LIN {X 0,Y 409.998,Z 362.021,A -85,B 0,C 180,E1 -10362.384,E2 -10362.384} C_VEL
LIN {X 0,Y 409.907,Z 362.961,A -85,B 0,C 180,E1 -10363.887,E2 -10363.887} C_VEL
LIN {X 0,Y 409.94,Z 362.921,A -85,B 0,C 180,E1 -10364.9,E2 -10364.9} C_VEL
LIN {X 0,Y 410.047,Z 362.009,A -85,B 0,C 180,E1 -10366.309,E2 -10366.309} C_VEL
LIN {X 0,Y 410.116,Z 361.339,A -85,B 0,C 180,E1 -10366.936,E2 -10366.936} C_VEL
LIN {X 0,Y 410.312,Z 358.576,A -85,B 0,C 180,E1 -10368.473,E2 -10368.473} C_VEL
LIN {X 0,Y 410.578,Z 355.393,A -85,B 0,C 180,E1 -10369.711,E2 -10369.711} C_VEL
LIN {X 0,Y 410.758,Z 352.823,A -85,B 0,C 180,E1 -10370.532,E2 -10370.532} C_VEL
LIN {X 0,Y 411.107,Z 347.629,A -85,B 0,C 180,E1 -10371.826,E2 -10371.826} C_VEL
LIN {X 0,Y 411.62,Z 341.02,A -85,B 0,C 180,E1 -10373.121,E2 -10373.121} C_VEL
LIN {X 0,Y 412.051,Z 334.444,A -85,B 0,C 180,E1 -10374.162,E2 -10374.162} C_VEL
LIN {X 0,Y 412.673,Z 326.386,A -85,B 0,C 180,E1 -10375.197,E2 -10375.197} C_VEL
LIN {X 0,Y 413.3,Z 315.956,A -85,B 0,C 180,E1 -10376.238,E2 -10376.238} C_VEL
LIN {X 0,Y 413.735,Z 307.563,A -85,B 0,C 180,E1 -10376.888,E2 -10376.888} C_VEL
LIN {X 0,Y 413.706,Z 301.383,A -85,B 0,C 180,E1 -10377.3,E2 -10377.3} C_VEL
LIN {X 0,Y 411.503,Z 290.548,A -85,B 0,C 180,E1 -10377.925,E2 -10377.925} C_VEL
LIN {X 0,Y 410.193,Z 285.02,A -85,B 0,C 180,E1 -10378.2,E2 -10378.2} C_VEL
LIN {X 0,Y 410.313,Z 281.535,A -85,B 0,C 180,E1 -10381.088,E2 -10381.088} C_VEL
LIN {X 0,Y 410.369,Z 277.277,A -85,B 0,C 180,E1 -10384.714,E2 -10384.714} C_VEL
LIN {X 0,Y 410.554,Z 273.44,A -85,B 0,C 180,E1 -10388.057,E2 -10388.057} C_VEL
LIN {X 0,Y 410.699,Z 269.952,A -85,B 0,C 180,E1 -10391.158,E2 -10391.158} C_VEL
LIN {X 0,Y 410.819,Z 266.266,A -85,B 0,C 180,E1 -10394.537,E2 -10394.537} C_VEL
LIN {X 0,Y 411.08,Z 266.09,A -85,B 0,C 180,E1 -10397.317,E2 -10397.317} C_VEL
LIN {X 0,Y 411.211,Z 266.076,A -85,B 0,C 180,E1 -10400.778,E2 -10400.778} C_VEL
LIN {X 0,Y 411.18,Z 266.082,A -85,B 0,C 180,E1 -10404.473,E2 -10404.473} C_VEL
LIN {X 0,Y 411.188,Z 266.079,A -85,B 0,C 180,E1 -10406.874,E2 -10406.874} C_VEL
LIN {X 0,Y 411.214,Z 266.077,A -85,B 0,C 180,E1 -10410.645,E2 -10410.645} C_VEL
LIN {X 0,Y 411.219,Z 266.075,A -85,B 0,C 180,E1 -10413.62,E2 -10413.62} C_VEL
LIN {X 0,Y 411.179,Z 266.08,A -85,B 0,C 180,E1 -10416.853,E2 -10416.853} C_VEL
LIN {X 0,Y 411.199,Z 266.078,A -85,B 0,C 180,E1 -10420.052,E2 -10420.052} C_VEL
LIN {X 0,Y 411.247,Z 266.07,A -85,B 0,C 180,E1 -10423.133,E2 -10423.133} C_VEL
LIN {X 0,Y 411.299,Z 266.064,A -85,B 0,C 180,E1 -10426.893,E2 -10426.893} C_VEL
LIN {X 0,Y 411.295,Z 266.063,A -85,B 0,C 180,E1 -10430.163,E2 -10430.163} C_VEL
LIN {X 0,Y 411.41,Z 266.047,A -85,B 0,C 180,E1 -10433.134,E2 -10433.134} C_VEL
LIN {X 0,Y 411.457,Z 266.044,A -85,B 0,C 180,E1 -10437.065,E2 -10437.065} C_VEL
LIN {X 0,Y 411.629,Z 266.022,A -85,B 0,C 180,E1 -10440.002,E2 -10440.002} C_VEL
LIN {X 0,Y 411.447,Z 266.044,A -85,B 0,C 180,E1 -10442.939,E2 -10442.939} C_VEL
LIN {X 0,Y 411.451,Z 266.044,A -85,B 0,C 180,E1 -10446.869,E2 -10446.869} C_VEL
LIN {X 0,Y 411.285,Z 266.066,A -85,B 0,C 180,E1 -10449.841,E2 -10449.841} C_VEL
LIN {X 0,Y 411.304,Z 266.065,A -85,B 0,C 180,E1 -10453.111,E2 -10453.111} C_VEL
LIN {X 0,Y 411.249,Z 266.071,A -85,B 0,C 180,E1 -10456.891,E2 -10456.891} C_VEL
LIN {X 0,Y 411.223,Z 266.075,A -85,B 0,C 180,E1 -10459.989,E2 -10459.989} C_VEL
LIN {X 0,Y 411.189,Z 266.08,A -85,B 0,C 180,E1 -10463.15,E2 -10463.15} C_VEL
LIN {X 0,Y 411.189,Z 266.081,A -85,B 0,C 180,E1 -10466.386,E2 -10466.386} C_VEL
LIN {X 0,Y 411.192,Z 266.081,A -85,B 0,C 180,E1 -10469.715,E2 -10469.715} C_VEL
LIN {X 0,Y 411.201,Z 266.08,A -85,B 0,C 180,E1 -10473.158,E2 -10473.158} C_VEL
LIN {X 0,Y 411.187,Z 266.081,A -85,B 0,C 180,E1 -10476.554,E2 -10476.554} C_VEL
LIN {X 0,Y 411.222,Z 266.075,A -85,B 0,C 180,E1 -10479.732,E2 -10479.732} C_VEL
LIN {X 0,Y 411.173,Z 266.083,A -85,B 0,C 180,E1 -10483.135,E2 -10483.135} C_VEL
LIN {X 0,Y 411.164,Z 266.082,A -85,B 0,C 180,E1 -10485.883,E2 -10485.883} C_VEL
LIN {X 0,Y 411.16,Z 266.085,A -85,B 0,C 180,E1 -10488.774,E2 -10488.774} C_VEL
LIN {X 0,Y 411.218,Z 266.113,A -85,B 0,C 180,E1 -10490.778,E2 -10490.778} C_VEL
LIN {X 0,Y 412.203,Z 271.693,A -85,B 0,C 180,E1 -10493.971,E2 -10493.971} C_VEL
LIN {X 0,Y 412.916,Z 276.371,A -85,B 0,C 180,E1 -10496.513,E2 -10496.513} C_VEL
LIN {X 0,Y 412.699,Z 280.103,A -85,B 0,C 180,E1 -10498.373,E2 -10498.373} C_VEL
LIN {X 0,Y 412.092,Z 286.591,A -85,B 0,C 180,E1 -10501.478,E2 -10501.478} C_VEL
LIN {X 0,Y 411.4,Z 294.979,A -85,B 0,C 180,E1 -10505.329,E2 -10505.329} C_VEL
LIN {X 0,Y 410.851,Z 303.168,A -85,B 0,C 180,E1 -10508.949,E2 -10508.949} C_VEL
LIN {X 0,Y 410.524,Z 311.551,A -85,B 0,C 180,E1 -10512.568,E2 -10512.568} C_VEL
LIN {X 0,Y 410.219,Z 319.243,A -85,B 0,C 180,E1 -10515.807,E2 -10515.807} C_VEL
LIN {X 0,Y 411.907,Z 330.548,A -85,B 0,C 180,E1 -10516.284,E2 -10516.284} C_VEL
LIN {X 0,Y 412.841,Z 341.087,A -85,B 0,C 180,E1 -10516.9,E2 -10516.9} C_VEL
LIN {X 0,Y 412.852,Z 349.045,A -85,B 0,C 180,E1 -10517.466,E2 -10517.466} C_VEL
LIN {X 0,Y 412.264,Z 357.493,A -85,B 0,C 180,E1 -10518.197,E2 -10518.197} C_VEL
LIN {X 0,Y 411.762,Z 365.475,A -85,B 0,C 180,E1 -10519.055,E2 -10519.055} C_VEL
LIN {X 0,Y 411.295,Z 372.086,A -85,B 0,C 180,E1 -10519.914,E2 -10519.914} C_VEL
LIN {X 0,Y 410.86,Z 378.38,A -85,B 0,C 180,E1 -10520.897,E2 -10520.897} C_VEL
LIN {X 0,Y 410.538,Z 383.622,A -85,B 0,C 180,E1 -10521.882,E2 -10521.882} C_VEL
LIN {X 0,Y 410.251,Z 388.968,A -85,B 0,C 180,E1 -10523.114,E2 -10523.114} C_VEL
LIN {X 0,Y 410.082,Z 392.428,A -85,B 0,C 180,E1 -10524.099,E2 -10524.099} C_VEL
LIN {X 0,Y 410.021,Z 396.434,A -85,B 0,C 180,E1 -10525.578,E2 -10525.578} C_VEL
LIN {X 0,Y 409.985,Z 399.189,A -85,B 0,C 180,E1 -10527.054,E2 -10527.054} C_VEL
LIN {X 0,Y 410.021,Z 400.293,A -85,B 0,C 180,E1 -10528.037,E2 -10528.037} C_VEL
LIN {X 0,Y 409.979,Z 400.923,A -85,B 0,C 180,E1 -10529.019,E2 -10529.019} C_VEL
LIN {X 0,Y 409.974,Z 401.092,A -85,B 0,C 180,E1 -10530.001,E2 -10530.001} C_VEL
LIN {X 0,Y 409.979,Z 400.763,A -85,B 0,C 180,E1 -10530.984,E2 -10530.984} C_VEL
LIN {X 0,Y 410.025,Z 399.839,A -85,B 0,C 180,E1 -10531.966,E2 -10531.966} C_VEL
LIN {X 0,Y 410.021,Z 398.414,A -85,B 0,C 180,E1 -10532.949,E2 -10532.949} C_VEL
LIN {X 0,Y 410.022,Z 395.317,A -85,B 0,C 180,E1 -10534.425,E2 -10534.425} C_VEL
LIN {X 0,Y 410.068,Z 390.877,A -85,B 0,C 180,E1 -10535.903,E2 -10535.903} C_VEL
LIN {X 0,Y 410.334,Z 385.927,A -85,B 0,C 180,E1 -10537.134,E2 -10537.134} C_VEL
LIN {X 0,Y 410.538,Z 379.661,A -85,B 0,C 180,E1 -10538.368,E2 -10538.368} C_VEL
LIN {X 0,Y 410.816,Z 373.538,A -85,B 0,C 180,E1 -10539.354,E2 -10539.354} C_VEL
LIN {X 0,Y 411.261,Z 366.093,A -85,B 0,C 180,E1 -10540.338,E2 -10540.338} C_VEL
LIN {X 0,Y 411.655,Z 358.104,A -85,B 0,C 180,E1 -10541.199,E2 -10541.199} C_VEL
LIN {X 0,Y 412.187,Z 348.138,A -85,B 0,C 180,E1 -10542.057,E2 -10542.057} C_VEL
LIN {X 0,Y 411.964,Z 338.649,A -85,B 0,C 180,E1 -10542.689,E2 -10542.689} C_VEL
LIN {X 0,Y 411.03,Z 328.221,A -85,B 0,C 180,E1 -10543.212,E2 -10543.212} C_VEL
LIN {X 0,Y 410.158,Z 319.531,A -85,B 0,C 180,E1 -10543.534,E2 -10543.534} C_VEL
LIN {X 0,Y 410.403,Z 311.332,A -85,B 0,C 180,E1 -10546.926,E2 -10546.926} C_VEL
LIN {X 0,Y 410.692,Z 302.714,A -85,B 0,C 180,E1 -10550.538,E2 -10550.538} C_VEL
LIN {X 0,Y 411.06,Z 295.284,A -85,B 0,C 180,E1 -10553.691,E2 -10553.691} C_VEL
LIN {X 0,Y 411.607,Z 286.782,A -85,B 0,C 180,E1 -10557.391,E2 -10557.391} C_VEL
LIN {X 0,Y 412.159,Z 279.227,A -85,B 0,C 180,E1 -10560.768,E2 -10560.768} C_VEL
LIN {X 0,Y 412.454,Z 273.561,A -85,B 0,C 180,E1 -10563.39,E2 -10563.39} C_VEL
LIN {X 0,Y 411.599,Z 268.219,A -85,B 0,C 180,E1 -10566.027,E2 -10566.027} C_VEL
LIN {X 0,Y 411.234,Z 266.075,A -85,B 0,C 180,E1 -10567.198,E2 -10567.198} C_VEL
LIN {X 0,Y 411.188,Z 266.079,A -85,B 0,C 180,E1 -10570.505,E2 -10570.505} C_VEL
LIN {X 0,Y 411.182,Z 266.078,A -85,B 0,C 180,E1 -10573.134,E2 -10573.134} C_VEL
LIN {X 0,Y 411.177,Z 266.082,A -85,B 0,C 180,E1 -10575.881,E2 -10575.881} C_VEL
LIN {X 0,Y 411.172,Z 266.079,A -85,B 0,C 180,E1 -10578.772,E2 -10578.772} C_VEL
LIN {X 0,Y 411.198,Z 266.079,A -85,B 0,C 180,E1 -10582.025,E2 -10582.025} C_VEL
LIN {X 0,Y 411.215,Z 266.078,A -85,B 0,C 180,E1 -10585.666,E2 -10585.666} C_VEL
LIN {X 0,Y 411.199,Z 266.078,A -85,B 0,C 180,E1 -10589.152,E2 -10589.152} C_VEL
LIN {X 0,Y 411.268,Z 266.067,A -85,B 0,C 180,E1 -10592.522,E2 -10592.522} C_VEL
LIN {X 0,Y 411.229,Z 266.074,A -85,B 0,C 180,E1 -10595.783,E2 -10595.783} C_VEL
LIN {X 0,Y 411.205,Z 266.079,A -85,B 0,C 180,E1 -10598.965,E2 -10598.965} C_VEL
LIN {X 0,Y 411.254,Z 266.069,A -85,B 0,C 180,E1 -10602.084,E2 -10602.084} C_VEL
LIN {X 0,Y 411.268,Z 266.071,A -85,B 0,C 180,E1 -10605.146,E2 -10605.146} C_VEL
LIN {X 0,Y 411.291,Z 266.065,A -85,B 0,C 180,E1 -10608.166,E2 -10608.166} C_VEL
LIN {X 0,Y 411.446,Z 266.046,A -85,B 0,C 180,E1 -10612.19,E2 -10612.19} C_VEL
LIN {X 0,Y 411.473,Z 266.043,A -85,B 0,C 180,E1 -10614.116,E2 -10614.116} C_VEL
LIN {X 0,Y 411.517,Z 266.037,A -85,B 0,C 180,E1 -10618.041,E2 -10618.041} C_VEL
LIN {X 0,Y 411.646,Z 266.021,A -85,B 0,C 180,E1 -10619.998,E2 -10619.998} C_VEL
LIN {X 0,Y 411.47,Z 266.044,A -85,B 0,C 180,E1 -10622.935,E2 -10622.935} C_VEL
LIN {X 0,Y 411.465,Z 266.045,A -85,B 0,C 180,E1 -10626.865,E2 -10626.865} C_VEL
LIN {X 0,Y 411.358,Z 266.058,A -85,B 0,C 180,E1 -10628.843,E2 -10628.843} C_VEL
LIN {X 0,Y 411.287,Z 266.067,A -85,B 0,C 180,E1 -10631.831,E2 -10631.831} C_VEL
LIN {X 0,Y 411.262,Z 266.069,A -85,B 0,C 180,E1 -10634.85,E2 -10634.85} C_VEL
LIN {X 0,Y 411.254,Z 266.072,A -85,B 0,C 180,E1 -10637.913,E2 -10637.913} C_VEL
LIN {X 0,Y 411.197,Z 266.076,A -85,B 0,C 180,E1 -10641.032,E2 -10641.032} C_VEL
LIN {X 0,Y 411.226,Z 266.075,A -85,B 0,C 180,E1 -10644.213,E2 -10644.213} C_VEL
LIN {X 0,Y 411.257,Z 266.072,A -85,B 0,C 180,E1 -10647.475,E2 -10647.475} C_VEL
LIN {X 0,Y 411.186,Z 266.077,A -85,B 0,C 180,E1 -10650.845,E2 -10650.845} C_VEL
LIN {X 0,Y 411.202,Z 266.076,A -85,B 0,C 180,E1 -10654.331,E2 -10654.331} C_VEL
LIN {X 0,Y 411.199,Z 266.078,A -85,B 0,C 180,E1 -10657.97,E2 -10657.97} C_VEL
LIN {X 0,Y 411.203,Z 266.079,A -85,B 0,C 180,E1 -10661.233,E2 -10661.233} C_VEL
LIN {X 0,Y 411.229,Z 266.073,A -85,B 0,C 180,E1 -10664.48,E2 -10664.48} C_VEL
LIN {X 0,Y 411.22,Z 266.077,A -85,B 0,C 180,E1 -10667.295,E2 -10667.295} C_VEL
LIN {X 0,Y 411.222,Z 266.076,A -85,B 0,C 180,E1 -10670.775,E2 -10670.775} C_VEL
LIN {X 0,Y 411.188,Z 266.078,A -85,B 0,C 180,E1 -10674.469,E2 -10674.469} C_VEL
LIN {X 0,Y 411.195,Z 266.08,A -85,B 0,C 180,E1 -10676.871,E2 -10676.871} C_VEL
LIN {X 0,Y 411.228,Z 266.076,A -85,B 0,C 180,E1 -10680.64,E2 -10680.64} C_VEL
LIN {X 0,Y 411.224,Z 266.073,A -85,B 0,C 180,E1 -10683.617,E2 -10683.617} C_VEL
LIN {X 0,Y 411.194,Z 266.079,A -85,B 0,C 180,E1 -10686.851,E2 -10686.851} C_VEL
LIN {X 0,Y 411.199,Z 266.078,A -85,B 0,C 180,E1 -10690.048,E2 -10690.048} C_VEL
LIN {X 0,Y 410.957,Z 266.107,A -85,B 0,C 180,E1 -10693.263,E2 -10693.263} C_VEL
LIN {X 0,Y 410.693,Z 266.143,A -85,B 0,C 180,E1 -10695.125,E2 -10695.125} C_VEL
LIN {X 0,Y 410.71,Z 268.309,A -85,B 0,C 180,E1 -10697.245,E2 -10697.245} C_VEL
LIN {X 0,Y 410.537,Z 272.981,A -85,B 0,C 180,E1 -10701.136,E2 -10701.136} C_VEL
LIN {X 0,Y 410.601,Z 275.356,A -85,B 0,C 180,E1 -10703.117,E2 -10703.117} C_VEL
LIN {X 0,Y 410.49,Z 278.995,A -85,B 0,C 180,E1 -10706.072,E2 -10706.072} C_VEL
LIN {X 0,Y 410.232,Z 282.687,A -85,B 0,C 180,E1 -10709.017,E2 -10709.017} C_VEL
LIN {X 0,Y 410.145,Z 284.671,A -85,B 0,C 180,E1 -10710.582,E2 -10710.582} C_VEL
LIN {X 0,Y 412.205,Z 296.714,A -85,B 0,C 180,E1 -10711.159,E2 -10711.159} C_VEL
LIN {X 0,Y 412.893,Z 302.077,A -85,B 0,C 180,E1 -10711.462,E2 -10711.462} C_VEL
LIN {X 0,Y 412.472,Z 312.617,A -85,B 0,C 180,E1 -10712.196,E2 -10712.196} C_VEL
LIN {X 0,Y 412.107,Z 320.89,A -85,B 0,C 180,E1 -10712.931,E2 -10712.931} C_VEL
LIN {X 0,Y 411.672,Z 328.745,A -85,B 0,C 180,E1 -10713.792,E2 -10713.792} C_VEL
LIN {X 0,Y 411.389,Z 335.207,A -85,B 0,C 180,E1 -10714.653,E2 -10714.653} C_VEL
LIN {X 0,Y 410.976,Z 341.39,A -85,B 0,C 180,E1 -10715.642,E2 -10715.642} C_VEL
LIN {X 0,Y 410.771,Z 347.667,A -85,B 0,C 180,E1 -10716.877,E2 -10716.877} C_VEL
LIN {X 0,Y 410.391,Z 353.532,A -85,B 0,C 180,E1 -10718.369,E2 -10718.369} C_VEL
LIN {X 0,Y 410.237,Z 356.577,A -85,B 0,C 180,E1 -10719.365,E2 -10719.365} C_VEL
LIN {X 0,Y 410.083,Z 359.907,A -85,B 0,C 180,E1 -10720.865,E2 -10720.865} C_VEL
LIN {X 0,Y 410.006,Z 361.951,A -85,B 0,C 180,E1 -10722.313,E2 -10722.313} C_VEL
LIN {X 0,Y 409.998,Z 362.021,A -85,B 0,C 180,E1 -10722.384,E2 -10722.384} C_VEL
LIN {X 0,Y 409.271,Z 362.759,A -85,B 0,C 180,E1 -10723.2,E2 -10723.2} C_VEL
LIN {X 0,Y 406.381,Z 363.211,A -85,B 0,C 180,E1 -10724.532,E2 -10724.532} C_VEL
LIN {X 0,Y 403.577,Z 362.803,A -85,B 0,C 180,E1 -10725.882,E2 -10725.882} C_VEL
LIN {X 0,Y 402.999,Z 361.972,A -85,B 0,C 180,E1 -10726.713,E2 -10726.713} C_VEL
LIN {X 0,Y 403.203,Z 359.617,A -85,B 0,C 180,E1 -10728.284,E2 -10728.284} C_VEL
LIN {X 0,Y 403.416,Z 357.245,A -85,B 0,C 180,E1 -10729.328,E2 -10729.328} C_VEL
LIN {X 0,Y 403.766,Z 352.366,A -85,B 0,C 180,E1 -10730.904,E2 -10730.904} C_VEL
LIN {X 0,Y 404.11,Z 348.209,A -85,B 0,C 180,E1 -10731.956,E2 -10731.956} C_VEL
LIN {X 0,Y 404.606,Z 342.156,A -85,B 0,C 180,E1 -10733.183,E2 -10733.183} C_VEL
LIN {X 0,Y 405.012,Z 336.926,A -85,B 0,C 180,E1 -10734.064,E2 -10734.064} C_VEL
LIN {X 0,Y 405.465,Z 330.348,A -85,B 0,C 180,E1 -10734.991,E2 -10734.991} C_VEL
LIN {X 0,Y 405.972,Z 323.212,A -85,B 0,C 180,E1 -10735.822,E2 -10735.822} C_VEL
LIN {X 0,Y 406.504,Z 315.296,A -85,B 0,C 180,E1 -10736.577,E2 -10736.577} C_VEL
LIN {X 0,Y 406.915,Z 307.924,A -85,B 0,C 180,E1 -10737.152,E2 -10737.152} C_VEL
LIN {X 0,Y 406.94,Z 302.908,A -85,B 0,C 180,E1 -10737.498,E2 -10737.498} C_VEL
LIN {X 0,Y 404.603,Z 291.351,A -85,B 0,C 180,E1 -10738.2,E2 -10738.2} C_VEL
LIN {X 0,Y 403.15,Z 285.374,A -85,B 0,C 180,E1 -10738.504,E2 -10738.504} C_VEL
LIN {X 0,Y 403.26,Z 281.77,A -85,B 0,C 180,E1 -10741.521,E2 -10741.521} C_VEL
LIN {X 0,Y 403.314,Z 277.633,A -85,B 0,C 180,E1 -10745.101,E2 -10745.101} C_VEL
LIN {X 0,Y 403.506,Z 273.912,A -85,B 0,C 180,E1 -10748.397,E2 -10748.397} C_VEL
LIN {X 0,Y 403.662,Z 270.44,A -85,B 0,C 180,E1 -10751.53,E2 -10751.53} C_VEL
LIN {X 0,Y 403.79,Z 267.269,A -85,B 0,C 180,E1 -10754.474,E2 -10754.474} C_VEL
LIN {X 0,Y 404.016,Z 266.97,A -85,B 0,C 180,E1 -10756.935,E2 -10756.935} C_VEL
LIN {X 0,Y 404.148,Z 266.956,A -85,B 0,C 180,E1 -10759.956,E2 -10759.956} C_VEL
LIN {X 0,Y 404.121,Z 266.961,A -85,B 0,C 180,E1 -10763.125,E2 -10763.125} C_VEL
LIN {X 0,Y 404.126,Z 266.96,A -85,B 0,C 180,E1 -10766.189,E2 -10766.189} C_VEL
LIN {X 0,Y 404.127,Z 266.957,A -85,B 0,C 180,E1 -10769.716,E2 -10769.716} C_VEL
LIN {X 0,Y 404.177,Z 266.951,A -85,B 0,C 180,E1 -10773.124,E2 -10773.124} C_VEL
LIN {X 0,Y 404.157,Z 266.956,A -85,B 0,C 180,E1 -10775.336,E2 -10775.336} C_VEL
LIN {X 0,Y 404.122,Z 266.958,A -85,B 0,C 180,E1 -10778.582,E2 -10778.582} C_VEL
LIN {X 0,Y 404.194,Z 266.949,A -85,B 0,C 180,E1 -10781.763,E2 -10781.763} C_VEL
LIN {X 0,Y 404.192,Z 266.95,A -85,B 0,C 180,E1 -10784.884,E2 -10784.884} C_VEL
LIN {X 0,Y 404.256,Z 266.945,A -85,B 0,C 180,E1 -10787.961,E2 -10787.961} C_VEL
LIN {X 0,Y 404.281,Z 266.939,A -85,B 0,C 180,E1 -10791.001,E2 -10791.001} C_VEL
LIN {X 0,Y 404.379,Z 266.923,A -85,B 0,C 180,E1 -10794.016,E2 -10794.016} C_VEL
LIN {X 0,Y 404.472,Z 266.912,A -85,B 0,C 180,E1 -10798.01,E2 -10798.01} C_VEL
LIN {X 0,Y 404.599,Z 266.898,A -85,B 0,C 180,E1 -10800.002,E2 -10800.002} C_VEL
LIN {X 0,Y 404.405,Z 266.921,A -85,B 0,C 180,E1 -10802.99,E2 -10802.99} C_VEL
LIN {X 0,Y 404.402,Z 266.923,A -85,B 0,C 180,E1 -10806.989,E2 -10806.989} C_VEL
LIN {X 0,Y 404.251,Z 266.944,A -85,B 0,C 180,E1 -10810.013,E2 -10810.013} C_VEL
LIN {X 0,Y 404.257,Z 266.943,A -85,B 0,C 180,E1 -10813.213,E2 -10813.213} C_VEL
LIN {X 0,Y 404.207,Z 266.948,A -85,B 0,C 180,E1 -10817.009,E2 -10817.009} C_VEL
LIN {X 0,Y 404.156,Z 266.953,A -85,B 0,C 180,E1 -10820.353,E2 -10820.353} C_VEL
LIN {X 0,Y 404.153,Z 266.954,A -85,B 0,C 180,E1 -10823.577,E2 -10823.577} C_VEL
LIN {X 0,Y 404.128,Z 266.959,A -85,B 0,C 180,E1 -10826.883,E2 -10826.883} C_VEL
LIN {X 0,Y 404.138,Z 266.959,A -85,B 0,C 180,E1 -10830.287,E2 -10830.287} C_VEL
LIN {X 0,Y 404.139,Z 266.963,A -85,B 0,C 180,E1 -10833.814,E2 -10833.814} C_VEL
LIN {X 0,Y 404.132,Z 266.961,A -85,B 0,C 180,E1 -10836.877,E2 -10836.877} C_VEL
LIN {X 0,Y 404.161,Z 266.956,A -85,B 0,C 180,E1 -10840.085,E2 -10840.085} C_VEL
LIN {X 0,Y 404.154,Z 266.957,A -85,B 0,C 180,E1 -10843.086,E2 -10843.086} C_VEL
LIN {X 0,Y 404.144,Z 266.956,A -85,B 0,C 180,E1 -10845.928,E2 -10845.928} C_VEL
LIN {X 0,Y 404.115,Z 266.963,A -85,B 0,C 180,E1 -10848.637,E2 -10848.637} C_VEL
LIN {X 0,Y 404.185,Z 267.016,A -85,B 0,C 180,E1 -10850.446,E2 -10850.446} C_VEL
LIN {X 0,Y 405.207,Z 272.822,A -85,B 0,C 180,E1 -10853.866,E2 -10853.866} C_VEL
LIN {X 0,Y 405.893,Z 277.333,A -85,B 0,C 180,E1 -10856.355,E2 -10856.355} C_VEL
LIN {X 0,Y 405.601,Z 281.932,A -85,B 0,C 180,E1 -10858.682,E2 -10858.682} C_VEL
LIN {X 0,Y 405.067,Z 287.708,A -85,B 0,C 180,E1 -10861.504,E2 -10861.504} C_VEL
LIN {X 0,Y 404.342,Z 295.939,A -85,B 0,C 180,E1 -10865.347,E2 -10865.347} C_VEL
LIN {X 0,Y 403.781,Z 304.226,A -85,B 0,C 180,E1 -10869.097,E2 -10869.097} C_VEL
LIN {X 0,Y 403.427,Z 312.579,A -85,B 0,C 180,E1 -10872.775,E2 -10872.775} C_VEL
LIN {X 0,Y 403.19,Z 318.864,A -85,B 0,C 180,E1 -10875.49,E2 -10875.49} C_VEL
LIN {X 0,Y 405.072,Z 331.754,A -85,B 0,C 180,E1 -10876.079,E2 -10876.079} C_VEL
LIN {X 0,Y 405.926,Z 341.516,A -85,B 0,C 180,E1 -10876.677,E2 -10876.677} C_VEL
LIN {X 0,Y 405.937,Z 349.273,A -85,B 0,C 180,E1 -10877.249,E2 -10877.249} C_VEL
LIN {X 0,Y 405.333,Z 357.62,A -85,B 0,C 180,E1 -10877.992,E2 -10877.992} C_VEL
LIN {X 0,Y 404.803,Z 365.524,A -85,B 0,C 180,E1 -10878.865,E2 -10878.865} C_VEL
LIN {X 0,Y 404.312,Z 372.071,A -85,B 0,C 180,E1 -10879.738,E2 -10879.738} C_VEL
LIN {X 0,Y 403.849,Z 378.313,A -85,B 0,C 180,E1 -10880.738,E2 -10880.738} C_VEL
LIN {X 0,Y 403.48,Z 383.508,A -85,B 0,C 180,E1 -10881.739,E2 -10881.739} C_VEL
LIN {X 0,Y 403.19,Z 388.81,A -85,B 0,C 180,E1 -10882.993,E2 -10882.993} C_VEL
LIN {X 0,Y 402.981,Z 393.763,A -85,B 0,C 180,E1 -10884.497,E2 -10884.497} C_VEL
LIN {X 0,Y 402.893,Z 397.281,A -85,B 0,C 180,E1 -10886,E2 -10886} C_VEL
LIN {X 0,Y 402.884,Z 398.926,A -85,B 0,C 180,E1 -10887.002,E2 -10887.002} C_VEL
LIN {X 0,Y 402.95,Z 400.003,A -85,B 0,C 180,E1 -10888.002,E2 -10888.002} C_VEL
LIN {X 0,Y 402.904,Z 400.606,A -85,B 0,C 180,E1 -10889.002,E2 -10889.002} C_VEL
LIN {X 0,Y 402.896,Z 400.749,A -85,B 0,C 180,E1 -10890.001,E2 -10890.001} C_VEL
LIN {X 0,Y 402.904,Z 400.407,A -85,B 0,C 180,E1 -10891.001,E2 -10891.001} C_VEL
LIN {X 0,Y 402.954,Z 399.47,A -85,B 0,C 180,E1 -10892,E2 -10892} C_VEL
LIN {X 0,Y 402.92,Z 398.016,A -85,B 0,C 180,E1 -10893.001,E2 -10893.001} C_VEL
LIN {X 0,Y 402.952,Z 394.891,A -85,B 0,C 180,E1 -10894.503,E2 -10894.503} C_VEL
LIN {X 0,Y 402.991,Z 390.392,A -85,B 0,C 180,E1 -10896.008,E2 -10896.008} C_VEL
LIN {X 0,Y 403.281,Z 385.394,A -85,B 0,C 180,E1 -10897.26,E2 -10897.26} C_VEL
LIN {X 0,Y 403.497,Z 379.08,A -85,B 0,C 180,E1 -10898.515,E2 -10898.515} C_VEL
LIN {X 0,Y 403.782,Z 372.902,A -85,B 0,C 180,E1 -10899.519,E2 -10899.519} C_VEL
LIN {X 0,Y 404.192,Z 366.42,A -85,B 0,C 180,E1 -10900.394,E2 -10900.394} C_VEL
LIN {X 0,Y 404.495,Z 359.793,A -85,B 0,C 180,E1 -10901.146,E2 -10901.146} C_VEL
LIN {X 0,Y 404.986,Z 351.783,A -85,B 0,C 180,E1 -10901.894,E2 -10901.894} C_VEL
LIN {X 0,Y 405.217,Z 343.667,A -85,B 0,C 180,E1 -10902.509,E2 -10902.509} C_VEL
LIN {X 0,Y 404.553,Z 334.884,A -85,B 0,C 180,E1 -10903.053,E2 -10903.053} C_VEL
LIN {X 0,Y 403.724,Z 325.792,A -85,B 0,C 180,E1 -10903.484,E2 -10903.484} C_VEL
LIN {X 0,Y 403.086,Z 319.207,A -85,B 0,C 180,E1 -10903.74,E2 -10903.74} C_VEL
LIN {X 0,Y 403.323,Z 310.929,A -85,B 0,C 180,E1 -10907.232,E2 -10907.232} C_VEL
LIN {X 0,Y 403.65,Z 302.331,A -85,B 0,C 180,E1 -10910.913,E2 -10910.913} C_VEL
LIN {X 0,Y 403.983,Z 296.148,A -85,B 0,C 180,E1 -10913.587,E2 -10913.587} C_VEL
LIN {X 0,Y 404.45,Z 288.78,A -85,B 0,C 180,E1 -10916.86,E2 -10916.86} C_VEL
LIN {X 0,Y 405.032,Z 281.362,A -85,B 0,C 180,E1 -10920.213,E2 -10920.213} C_VEL
LIN {X 0,Y 405.448,Z 275.249,A -85,B 0,C 180,E1 -10923.081,E2 -10923.081} C_VEL
LIN {X 0,Y 404.836,Z 270.727,A -85,B 0,C 180,E1 -10925.32,E2 -10925.32} C_VEL
LIN {X 0,Y 404.171,Z 266.955,A -85,B 0,C 180,E1 -10927.323,E2 -10927.323} C_VEL
LIN {X 0,Y 404.157,Z 266.957,A -85,B 0,C 180,E1 -10930.08,E2 -10930.08} C_VEL
LIN {X 0,Y 404.162,Z 266.952,A -85,B 0,C 180,E1 -10933.084,E2 -10933.084} C_VEL
LIN {X 0,Y 404.157,Z 266.956,A -85,B 0,C 180,E1 -10935.926,E2 -10935.926} C_VEL
LIN {X 0,Y 404.127,Z 266.957,A -85,B 0,C 180,E1 -10938.635,E2 -10938.635} C_VEL
LIN {X 0,Y 404.157,Z 266.956,A -85,B 0,C 180,E1 -10941.493,E2 -10941.493} C_VEL
LIN {X 0,Y 404.193,Z 266.949,A -85,B 0,C 180,E1 -10944.983,E2 -10944.983} C_VEL
LIN {X 0,Y 404.151,Z 266.954,A -85,B 0,C 180,E1 -10948.553,E2 -10948.553} C_VEL
LIN {X 0,Y 404.205,Z 266.948,A -85,B 0,C 180,E1 -10952,E2 -10952} C_VEL
LIN {X 0,Y 404.183,Z 266.953,A -85,B 0,C 180,E1 -10955.333,E2 -10955.333} C_VEL
LIN {X 0,Y 404.147,Z 266.954,A -85,B 0,C 180,E1 -10958.58,E2 -10958.58} C_VEL
LIN {X 0,Y 404.213,Z 266.947,A -85,B 0,C 180,E1 -10961.761,E2 -10961.761} C_VEL
LIN {X 0,Y 404.214,Z 266.949,A -85,B 0,C 180,E1 -10964.881,E2 -10964.881} C_VEL
LIN {X 0,Y 404.264,Z 266.94,A -85,B 0,C 180,E1 -10967.957,E2 -10967.957} C_VEL
LIN {X 0,Y 404.273,Z 266.942,A -85,B 0,C 180,E1 -10970.997,E2 -10970.997} C_VEL
LIN {X 0,Y 404.42,Z 266.921,A -85,B 0,C 180,E1 -10974.013,E2 -10974.013} C_VEL
LIN {X 0,Y 404.486,Z 266.913,A -85,B 0,C 180,E1 -10978.007,E2 -10978.007} C_VEL
LIN {X 0,Y 404.615,Z 266.897,A -85,B 0,C 180,E1 -10979.998,E2 -10979.998} C_VEL
LIN {X 0,Y 404.427,Z 266.921,A -85,B 0,C 180,E1 -10982.986,E2 -10982.986} C_VEL
LIN {X 0,Y 404.416,Z 266.922,A -85,B 0,C 180,E1 -10986.985,E2 -10986.985} C_VEL
LIN {X 0,Y 404.262,Z 266.942,A -85,B 0,C 180,E1 -10990.01,E2 -10990.01} C_VEL
LIN {X 0,Y 404.269,Z 266.939,A -85,B 0,C 180,E1 -10993.209,E2 -10993.209} C_VEL
LIN {X 0,Y 404.218,Z 266.946,A -85,B 0,C 180,E1 -10997.005,E2 -10997.005} C_VEL
LIN {X 0,Y 404.164,Z 266.954,A -85,B 0,C 180,E1 -11000.349,E2 -11000.349} C_VEL
LIN {X 0,Y 404.169,Z 266.955,A -85,B 0,C 180,E1 -11003.572,E2 -11003.572} C_VEL
LIN {X 0,Y 404.183,Z 266.953,A -85,B 0,C 180,E1 -11005.764,E2 -11005.764} C_VEL
LIN {X 0,Y 404.193,Z 266.952,A -85,B 0,C 180,E1 -11007.997,E2 -11007.997} C_VEL
LIN {X 0,Y 404.136,Z 266.959,A -85,B 0,C 180,E1 -11011.555,E2 -11011.555} C_VEL
LIN {X 0,Y 404.181,Z 266.951,A -85,B 0,C 180,E1 -11015.013,E2 -11015.013} C_VEL
LIN {X 0,Y 404.157,Z 266.954,A -85,B 0,C 180,E1 -11018.753,E2 -11018.753} C_VEL
LIN {X 0,Y 404.185,Z 266.952,A -85,B 0,C 180,E1 -11021.608,E2 -11021.608} C_VEL
LIN {X 0,Y 404.193,Z 266.949,A -85,B 0,C 180,E1 -11024.528,E2 -11024.528} C_VEL
LIN {X 0,Y 404.198,Z 266.952,A -85,B 0,C 180,E1 -11027.302,E2 -11027.302} C_VEL
LIN {X 0,Y 404.159,Z 266.953,A -85,B 0,C 180,E1 -11029.953,E2 -11029.953} C_VEL
LIN {X 0,Y 404.13,Z 266.96,A -85,B 0,C 180,E1 -11033.122,E2 -11033.122} C_VEL
LIN {X 0,Y 404.133,Z 266.956,A -85,B 0,C 180,E1 -11036.185,E2 -11036.185} C_VEL
LIN {X 0,Y 404.141,Z 266.955,A -85,B 0,C 180,E1 -11039.713,E2 -11039.713} C_VEL
LIN {X 0,Y 404.182,Z 266.953,A -85,B 0,C 180,E1 -11043.121,E2 -11043.121} C_VEL
LIN {X 0,Y 404.158,Z 266.956,A -85,B 0,C 180,E1 -11046.424,E2 -11046.424} C_VEL
LIN {X 0,Y 404.176,Z 266.951,A -85,B 0,C 180,E1 -11049.872,E2 -11049.872} C_VEL
LIN {X 0,Y 403.936,Z 266.982,A -85,B 0,C 180,E1 -11053.114,E2 -11053.114} C_VEL
LIN {X 0,Y 403.695,Z 267.015,A -85,B 0,C 180,E1 -11054.861,E2 -11054.861} C_VEL
LIN {X 0,Y 403.59,Z 267.449,A -85,B 0,C 180,E1 -11055.888,E2 -11055.888} C_VEL
LIN {X 0,Y 403.615,Z 269.862,A -85,B 0,C 180,E1 -11057.938,E2 -11057.938} C_VEL
LIN {X 0,Y 403.477,Z 274.641,A -85,B 0,C 180,E1 -11061.989,E2 -11061.989} C_VEL
LIN {X 0,Y 403.437,Z 277.065,A -85,B 0,C 180,E1 -11063.999,E2 -11063.999} C_VEL
LIN {X 0,Y 403.37,Z 280.737,A -85,B 0,C 180,E1 -11067.003,E2 -11067.003} C_VEL
LIN {X 0,Y 403.081,Z 284.998,A -85,B 0,C 180,E1 -11070.405,E2 -11070.405} C_VEL
LIN {X 0,Y 404.985,Z 296.22,A -85,B 0,C 180,E1 -11070.931,E2 -11070.931} C_VEL
LIN {X 0,Y 405.88,Z 301.578,A -85,B 0,C 180,E1 -11071.239,E2 -11071.239} C_VEL
LIN {X 0,Y 405.515,Z 312.327,A -85,B 0,C 180,E1 -11071.985,E2 -11071.985} C_VEL
LIN {X 0,Y 405.131,Z 320.711,A -85,B 0,C 180,E1 -11072.733,E2 -11072.733} C_VEL
LIN {X 0,Y 404.668,Z 328.654,A -85,B 0,C 180,E1 -11073.608,E2 -11073.608} C_VEL
LIN {X 0,Y 404.357,Z 335.188,A -85,B 0,C 180,E1 -11074.485,E2 -11074.485} C_VEL
LIN {X 0,Y 403.945,Z 341.426,A -85,B 0,C 180,E1 -11075.49,E2 -11075.49} C_VEL
LIN {X 0,Y 403.808,Z 346.491,A -85,B 0,C 180,E1 -11076.478,E2 -11076.478} C_VEL
LIN {X 0,Y 403.546,Z 350.692,A -85,B 0,C 180,E1 -11077.454,E2 -11077.454} C_VEL
LIN {X 0,Y 403.283,Z 354.47,A -85,B 0,C 180,E1 -11078.517,E2 -11078.517} C_VEL
LIN {X 0,Y 403.055,Z 358.568,A -85,B 0,C 180,E1 -11080.04,E2 -11080.04} C_VEL
LIN {X 0,Y 402.999,Z 360.563,A -85,B 0,C 180,E1 -11081.058,E2 -11081.058} C_VEL
LIN {X 0,Y 402.91,Z 362.326,A -85,B 0,C 180,E1 -11082.376,E2 -11082.376} C_VEL
LIN {X 0,Y 402.867,Z 363,A -85,B 0,C 180,E1 -11083.106,E2 -11083.106} C_VEL
LIN {X 0,Y 402.828,Z 363.36,A -85,B 0,C 180,E1 -11084.136,E2 -11084.136} C_VEL
LIN {X 0,Y 402.864,Z 363.19,A -85,B 0,C 180,E1 -11085.168,E2 -11085.168} C_VEL
LIN {X 0,Y 402.999,Z 361.972,A -85,B 0,C 180,E1 -11086.713,E2 -11086.713} C_VEL
LIN {X 0,Y 402.45,Z 360.936,A -85,B 0,C 180,E1 -11087.537,E2 -11087.537} C_VEL
LIN {X 0,Y 399.821,Z 358.726,A -85,B 0,C 180,E1 -11088.87,E2 -11088.87} C_VEL
LIN {X 0,Y 397.226,Z 355.629,A -85,B 0,C 180,E1 -11090.176,E2 -11090.176} C_VEL
LIN {X 0,Y 396.735,Z 353.141,A -85,B 0,C 180,E1 -11090.948,E2 -11090.948} C_VEL
LIN {X 0,Y 397.105,Z 348.793,A -85,B 0,C 180,E1 -11092.09,E2 -11092.09} C_VEL
LIN {X 0,Y 397.57,Z 343.589,A -85,B 0,C 180,E1 -11093.195,E2 -11093.195} C_VEL
LIN {X 0,Y 398.053,Z 337.637,A -85,B 0,C 180,E1 -11094.235,E2 -11094.235} C_VEL
LIN {X 0,Y 398.611,Z 330.074,A -85,B 0,C 180,E1 -11095.311,E2 -11095.311} C_VEL
LIN {X 0,Y 399.153,Z 323.217,A -85,B 0,C 180,E1 -11096.114,E2 -11096.114} C_VEL
LIN {X 0,Y 399.732,Z 314.812,A -85,B 0,C 180,E1 -11096.917,E2 -11096.917} C_VEL
LIN {X 0,Y 400.209,Z 306.963,A -85,B 0,C 180,E1 -11097.52,E2 -11097.52} C_VEL
LIN {X 0,Y 399.893,Z 302.926,A -85,B 0,C 180,E1 -11097.818,E2 -11097.818} C_VEL
LIN {X 0,Y 397.52,Z 291.5,A -85,B 0,C 180,E1 -11098.523,E2 -11098.523} C_VEL
LIN {X 0,Y 396.122,Z 285.671,A -85,B 0,C 180,E1 -11098.838,E2 -11098.838} C_VEL
LIN {X 0,Y 396.196,Z 281.792,A -85,B 0,C 180,E1 -11102.15,E2 -11102.15} C_VEL
LIN {X 0,Y 396.288,Z 277.626,A -85,B 0,C 180,E1 -11105.818,E2 -11105.818} C_VEL
LIN {X 0,Y 396.461,Z 274.363,A -85,B 0,C 180,E1 -11108.746,E2 -11108.746} C_VEL
LIN {X 0,Y 396.613,Z 270.936,A -85,B 0,C 180,E1 -11111.91,E2 -11111.91} C_VEL
LIN {X 0,Y 396.779,Z 267.874,A -85,B 0,C 180,E1 -11114.89,E2 -11114.89} C_VEL
LIN {X 0,Y 397.006,Z 267.847,A -85,B 0,C 180,E1 -11118.028,E2 -11118.028} C_VEL
LIN {X 0,Y 397.118,Z 267.835,A -85,B 0,C 180,E1 -11121.138,E2 -11121.138} C_VEL
LIN {X 0,Y 397.101,Z 267.836,A -85,B 0,C 180,E1 -11124.498,E2 -11124.498} C_VEL
LIN {X 0,Y 397.059,Z 267.839,A -85,B 0,C 180,E1 -11127.93,E2 -11127.93} C_VEL
LIN {X 0,Y 397.103,Z 267.831,A -85,B 0,C 180,E1 -11131.458,E2 -11131.458} C_VEL
LIN {X 0,Y 397.135,Z 267.828,A -85,B 0,C 180,E1 -11134.489,E2 -11134.489} C_VEL
LIN {X 0,Y 397.079,Z 267.837,A -85,B 0,C 180,E1 -11138.183,E2 -11138.183} C_VEL
LIN {X 0,Y 397.146,Z 267.829,A -85,B 0,C 180,E1 -11141.428,E2 -11141.428} C_VEL
LIN {X 0,Y 397.165,Z 267.827,A -85,B 0,C 180,E1 -11144.61,E2 -11144.61} C_VEL
LIN {X 0,Y 397.215,Z 267.82,A -85,B 0,C 180,E1 -11147.744,E2 -11147.744} C_VEL
LIN {X 0,Y 397.243,Z 267.814,A -85,B 0,C 180,E1 -11150.84,E2 -11150.84} C_VEL
LIN {X 0,Y 397.331,Z 267.8,A -85,B 0,C 180,E1 -11153.91,E2 -11153.91} C_VEL
LIN {X 0,Y 397.441,Z 267.787,A -85,B 0,C 180,E1 -11157.975,E2 -11157.975} C_VEL
LIN {X 0,Y 397.568,Z 267.774,A -85,B 0,C 180,E1 -11160.002,E2 -11160.002} C_VEL
LIN {X 0,Y 397.365,Z 267.798,A -85,B 0,C 180,E1 -11163.043,E2 -11163.043} C_VEL
LIN {X 0,Y 397.354,Z 267.802,A -85,B 0,C 180,E1 -11167.114,E2 -11167.114} C_VEL
LIN {X 0,Y 397.211,Z 267.823,A -85,B 0,C 180,E1 -11170.193,E2 -11170.193} C_VEL
LIN {X 0,Y 397.218,Z 267.821,A -85,B 0,C 180,E1 -11173.323,E2 -11173.323} C_VEL
LIN {X 0,Y 397.174,Z 267.823,A -85,B 0,C 180,E1 -11177.157,E2 -11177.157} C_VEL
LIN {X 0,Y 397.095,Z 267.833,A -85,B 0,C 180,E1 -11180.732,E2 -11180.732} C_VEL
LIN {X 0,Y 397.116,Z 267.832,A -85,B 0,C 180,E1 -11184.021,E2 -11184.021} C_VEL
LIN {X 0,Y 397.095,Z 267.837,A -85,B 0,C 180,E1 -11187.399,E2 -11187.399} C_VEL
LIN {X 0,Y 397.072,Z 267.843,A -85,B 0,C 180,E1 -11190.884,E2 -11190.884} C_VEL
LIN {X 0,Y 397.12,Z 267.834,A -85,B 0,C 180,E1 -11194.495,E2 -11194.495} C_VEL
LIN {X 0,Y 397.102,Z 267.835,A -85,B 0,C 180,E1 -11198.276,E2 -11198.276} C_VEL
LIN {X 0,Y 397.108,Z 267.832,A -85,B 0,C 180,E1 -11200.908,E2 -11200.908} C_VEL
LIN {X 0,Y 397.098,Z 267.837,A -85,B 0,C 180,E1 -11203.65,E2 -11203.65} C_VEL
LIN {X 0,Y 397.099,Z 267.833,A -85,B 0,C 180,E1 -11206.523,E2 -11206.523} C_VEL
LIN {X 0,Y 397.157,Z 267.921,A -85,B 0,C 180,E1 -11210.113,E2 -11210.113} C_VEL
LIN {X 0,Y 397.999,Z 272.869,A -85,B 0,C 180,E1 -11213.105,E2 -11213.105} C_VEL
LIN {X 0,Y 398.82,Z 277.785,A -85,B 0,C 180,E1 -11215.919,E2 -11215.919} C_VEL
LIN {X 0,Y 398.812,Z 281.275,A -85,B 0,C 180,E1 -11217.767,E2 -11217.767} C_VEL
LIN {X 0,Y 398.164,Z 287.654,A -85,B 0,C 180,E1 -11220.963,E2 -11220.963} C_VEL
LIN {X 0,Y 397.354,Z 295.821,A -85,B 0,C 180,E1 -11224.883,E2 -11224.883} C_VEL
LIN {X 0,Y 396.829,Z 302.9,A -85,B 0,C 180,E1 -11228.168,E2 -11228.168} C_VEL
LIN {X 0,Y 396.42,Z 311.214,A -85,B 0,C 180,E1 -11231.927,E2 -11231.927} C_VEL
LIN {X 0,Y 396.109,Z 318.493,A -85,B 0,C 180,E1 -11235.159,E2 -11235.159} C_VEL
LIN {X 0,Y 398.087,Z 331.452,A -85,B 0,C 180,E1 -11235.777,E2 -11235.777} C_VEL
LIN {X 0,Y 398.912,Z 340.497,A -85,B 0,C 180,E1 -11236.338,E2 -11236.338} C_VEL
LIN {X 0,Y 399.08,Z 348.029,A -85,B 0,C 180,E1 -11236.897,E2 -11236.897} C_VEL
LIN {X 0,Y 398.565,Z 356.528,A -85,B 0,C 180,E1 -11237.656,E2 -11237.656} C_VEL
LIN {X 0,Y 397.924,Z 364.553,A -85,B 0,C 180,E1 -11238.541,E2 -11238.541} C_VEL
LIN {X 0,Y 397.422,Z 370.352,A -85,B 0,C 180,E1 -11239.301,E2 -11239.301} C_VEL
LIN {X 0,Y 396.952,Z 376.823,A -85,B 0,C 180,E1 -11240.318,E2 -11240.318} C_VEL
LIN {X 0,Y 396.525,Z 382.217,A -85,B 0,C 180,E1 -11241.337,E2 -11241.337} C_VEL
LIN {X 0,Y 396.227,Z 386.733,A -85,B 0,C 180,E1 -11242.357,E2 -11242.357} C_VEL
LIN {X 0,Y 395.947,Z 391.542,A -85,B 0,C 180,E1 -11243.721,E2 -11243.721} C_VEL
LIN {X 0,Y 395.9,Z 394.814,A -85,B 0,C 180,E1 -11244.909,E2 -11244.909} C_VEL
LIN {X 0,Y 395.819,Z 397.027,A -85,B 0,C 180,E1 -11245.929,E2 -11245.929} C_VEL
LIN {X 0,Y 395.784,Z 398.665,A -85,B 0,C 180,E1 -11246.948,E2 -11246.948} C_VEL
LIN {X 0,Y 395.861,Z 399.717,A -85,B 0,C 180,E1 -11247.966,E2 -11247.966} C_VEL
LIN {X 0,Y 395.831,Z 400.291,A -85,B 0,C 180,E1 -11248.984,E2 -11248.984} C_VEL
LIN {X 0,Y 395.821,Z 400.404,A -85,B 0,C 180,E1 -11250.001,E2 -11250.001} C_VEL
LIN {X 0,Y 395.832,Z 400.044,A -85,B 0,C 180,E1 -11251.019,E2 -11251.019} C_VEL
LIN {X 0,Y 395.885,Z 399.095,A -85,B 0,C 180,E1 -11252.036,E2 -11252.036} C_VEL
LIN {X 0,Y 395.802,Z 396.753,A -85,B 0,C 180,E1 -11253.564,E2 -11253.564} C_VEL
LIN {X 0,Y 395.901,Z 393.059,A -85,B 0,C 180,E1 -11255.094,E2 -11255.094} C_VEL
LIN {X 0,Y 396.03,Z 388.151,A -85,B 0,C 180,E1 -11256.574,E2 -11256.574} C_VEL
LIN {X 0,Y 396.221,Z 383.652,A -85,B 0,C 180,E1 -11257.646,E2 -11257.646} C_VEL
LIN {X 0,Y 396.441,Z 378.479,A -85,B 0,C 180,E1 -11258.668,E2 -11258.668} C_VEL
LIN {X 0,Y 396.765,Z 372.248,A -85,B 0,C 180,E1 -11259.689,E2 -11259.689} C_VEL
LIN {X 0,Y 397.193,Z 365.702,A -85,B 0,C 180,E1 -11260.579,E2 -11260.579} C_VEL
LIN {X 0,Y 397.534,Z 358.998,A -85,B 0,C 180,E1 -11261.344,E2 -11261.344} C_VEL
LIN {X 0,Y 398.022,Z 350.883,A -85,B 0,C 180,E1 -11262.105,E2 -11262.105} C_VEL
LIN {X 0,Y 398.191,Z 344.926,A -85,B 0,C 180,E1 -11262.576,E2 -11262.576} C_VEL
LIN {X 0,Y 397.569,Z 335.721,A -85,B 0,C 180,E1 -11263.176,E2 -11263.176} C_VEL
LIN {X 0,Y 396.736,Z 326.453,A -85,B 0,C 180,E1 -11263.638,E2 -11263.638} C_VEL
LIN {X 0,Y 395.979,Z 318.939,A -85,B 0,C 180,E1 -11263.92,E2 -11263.92} C_VEL
LIN {X 0,Y 396.233,Z 312.491,A -85,B 0,C 180,E1 -11266.702,E2 -11266.702} C_VEL
LIN {X 0,Y 396.557,Z 303.174,A -85,B 0,C 180,E1 -11270.761,E2 -11270.761} C_VEL
LIN {X 0,Y 396.952,Z 295.812,A -85,B 0,C 180,E1 -11274.031,E2 -11274.031} C_VEL
LIN {X 0,Y 397.471,Z 288.422,A -85,B 0,C 180,E1 -11277.371,E2 -11277.371} C_VEL
LIN {X 0,Y 398.097,Z 281.047,A -85,B 0,C 180,E1 -11280.796,E2 -11280.796} C_VEL
LIN {X 0,Y 398.414,Z 276.116,A -85,B 0,C 180,E1 -11283.152,E2 -11283.152} C_VEL
LIN {X 0,Y 397.723,Z 271.157,A -85,B 0,C 180,E1 -11285.672,E2 -11285.672} C_VEL
LIN {X 0,Y 397.148,Z 267.829,A -85,B 0,C 180,E1 -11287.491,E2 -11287.491} C_VEL
LIN {X 0,Y 397.097,Z 267.832,A -85,B 0,C 180,E1 -11290.909,E2 -11290.909} C_VEL
LIN {X 0,Y 397.11,Z 267.833,A -85,B 0,C 180,E1 -11293.649,E2 -11293.649} C_VEL
LIN {X 0,Y 397.111,Z 267.831,A -85,B 0,C 180,E1 -11296.521,E2 -11296.521} C_VEL
LIN {X 0,Y 397.121,Z 267.83,A -85,B 0,C 180,E1 -11300.422,E2 -11300.422} C_VEL
LIN {X 0,Y 397.117,Z 267.831,A -85,B 0,C 180,E1 -11304.265,E2 -11304.265} C_VEL
LIN {X 0,Y 397.124,Z 267.829,A -85,B 0,C 180,E1 -11306.727,E2 -11306.727} C_VEL
LIN {X 0,Y 397.134,Z 267.828,A -85,B 0,C 180,E1 -11310.295,E2 -11310.295} C_VEL
LIN {X 0,Y 397.204,Z 267.819,A -85,B 0,C 180,E1 -11312.609,E2 -11312.609} C_VEL
LIN {X 0,Y 397.138,Z 267.828,A -85,B 0,C 180,E1 -11315.981,E2 -11315.981} C_VEL
LIN {X 0,Y 397.148,Z 267.827,A -85,B 0,C 180,E1 -11319.704,E2 -11319.704} C_VEL
LIN {X 0,Y 397.191,Z 267.823,A -85,B 0,C 180,E1 -11322.844,E2 -11322.844} C_VEL
LIN {X 0,Y 397.237,Z 267.817,A -85,B 0,C 180,E1 -11326.701,E2 -11326.701} C_VEL
LIN {X 0,Y 397.224,Z 267.817,A -85,B 0,C 180,E1 -11329.807,E2 -11329.807} C_VEL
LIN {X 0,Y 397.341,Z 267.806,A -85,B 0,C 180,E1 -11332.886,E2 -11332.886} C_VEL
LIN {X 0,Y 397.257,Z 267.816,A -85,B 0,C 180,E1 -11334.923,E2 -11334.923} C_VEL
LIN {X 0,Y 397.455,Z 267.788,A -85,B 0,C 180,E1 -11337.972,E2 -11337.972} C_VEL
LIN {X 0,Y 397.585,Z 267.772,A -85,B 0,C 180,E1 -11339.998,E2 -11339.998} C_VEL
LIN {X 0,Y 397.386,Z 267.797,A -85,B 0,C 180,E1 -11343.039,E2 -11343.039} C_VEL
LIN {X 0,Y 397.369,Z 267.799,A -85,B 0,C 180,E1 -11347.11,E2 -11347.11} C_VEL
LIN {X 0,Y 397.222,Z 267.821,A -85,B 0,C 180,E1 -11350.189,E2 -11350.189} C_VEL
LIN {X 0,Y 397.23,Z 267.816,A -85,B 0,C 180,E1 -11353.319,E2 -11353.319} C_VEL
LIN {X 0,Y 397.184,Z 267.822,A -85,B 0,C 180,E1 -11357.153,E2 -11357.153} C_VEL
LIN {X 0,Y 397.103,Z 267.832,A -85,B 0,C 180,E1 -11360.728,E2 -11360.728} C_VEL
LIN {X 0,Y 397.132,Z 267.832,A -85,B 0,C 180,E1 -11364.016,E2 -11364.016} C_VEL
LIN {X 0,Y 397.193,Z 267.822,A -85,B 0,C 180,E1 -11367.388,E2 -11367.388} C_VEL
LIN {X 0,Y 397.075,Z 267.835,A -85,B 0,C 180,E1 -11370.88,E2 -11370.88} C_VEL
LIN {X 0,Y 397.121,Z 267.829,A -85,B 0,C 180,E1 -11374.491,E2 -11374.491} C_VEL
LIN {X 0,Y 397.104,Z 267.832,A -85,B 0,C 180,E1 -11378.272,E2 -11378.272} C_VEL
LIN {X 0,Y 397.15,Z 267.827,A -85,B 0,C 180,E1 -11381.991,E2 -11381.991} C_VEL
LIN {X 0,Y 397.142,Z 267.83,A -85,B 0,C 180,E1 -11385.057,E2 -11385.057} C_VEL
LIN {X 0,Y 397.147,Z 267.826,A -85,B 0,C 180,E1 -11388.004,E2 -11388.004} C_VEL
LIN {X 0,Y 397.1,Z 267.832,A -85,B 0,C 180,E1 -11391.723,E2 -11391.723} C_VEL
LIN {X 0,Y 397.114,Z 267.831,A -85,B 0,C 180,E1 -11395.504,E2 -11395.504} C_VEL
LIN {X 0,Y 397.072,Z 267.839,A -85,B 0,C 180,E1 -11399.116,E2 -11399.116} C_VEL
LIN {X 0,Y 397.181,Z 267.825,A -85,B 0,C 180,E1 -11402.608,E2 -11402.608} C_VEL
LIN {X 0,Y 397.12,Z 267.83,A -85,B 0,C 180,E1 -11405.98,E2 -11405.98} C_VEL
LIN {X 0,Y 397.13,Z 267.828,A -85,B 0,C 180,E1 -11409.7,E2 -11409.7} C_VEL
LIN {X 0,Y 396.896,Z 267.859,A -85,B 0,C 180,E1 -11412.969,E2 -11412.969} C_VEL
LIN {X 0,Y 396.528,Z 267.908,A -85,B 0,C 180,E1 -11415.632,E2 -11415.632} C_VEL
LIN {X 0,Y 396.549,Z 270.302,A -85,B 0,C 180,E1 -11417.72,E2 -11417.72} C_VEL
LIN {X 0,Y 396.398,Z 275.132,A -85,B 0,C 180,E1 -11421.845,E2 -11421.845} C_VEL
LIN {X 0,Y 396.389,Z 277.562,A -85,B 0,C 180,E1 -11423.892,E2 -11423.892} C_VEL
LIN {X 0,Y 396.298,Z 281.272,A -85,B 0,C 180,E1 -11426.949,E2 -11426.949} C_VEL
LIN {X 0,Y 396.033,Z 285.499,A -85,B 0,C 180,E1 -11430.221,E2 -11430.221} C_VEL
LIN {X 0,Y 397.966,Z 296.776,A -85,B 0,C 180,E1 -11430.758,E2 -11430.758} C_VEL
LIN {X 0,Y 398.916,Z 303.091,A -85,B 0,C 180,E1 -11431.134,E2 -11431.134} C_VEL
LIN {X 0,Y 398.583,Z 312.03,A -85,B 0,C 180,E1 -11431.767,E2 -11431.767} C_VEL
LIN {X 0,Y 398.182,Z 320.525,A -85,B 0,C 180,E1 -11432.528,E2 -11432.528} C_VEL
LIN {X 0,Y 397.681,Z 328.56,A -85,B 0,C 180,E1 -11433.418,E2 -11433.418} C_VEL
LIN {X 0,Y 397.33,Z 335.17,A -85,B 0,C 180,E1 -11434.31,E2 -11434.31} C_VEL
LIN {X 0,Y 396.932,Z 341.458,A -85,B 0,C 180,E1 -11435.332,E2 -11435.332} C_VEL
LIN {X 0,Y 396.759,Z 346.584,A -85,B 0,C 180,E1 -11436.339,E2 -11436.339} C_VEL
LIN {X 0,Y 396.415,Z 351.983,A -85,B 0,C 180,E1 -11437.64,E2 -11437.64} C_VEL
LIN {X 0,Y 396.195,Z 355.406,A -85,B 0,C 180,E1 -11438.671,E2 -11438.671} C_VEL
LIN {X 0,Y 396.031,Z 358.19,A -85,B 0,C 180,E1 -11439.704,E2 -11439.704} C_VEL
LIN {X 0,Y 395.886,Z 361.223,A -85,B 0,C 180,E1 -11441.26,E2 -11441.26} C_VEL
LIN {X 0,Y 395.818,Z 362.704,A -85,B 0,C 180,E1 -11442.444,E2 -11442.444} C_VEL
LIN {X 0,Y 395.772,Z 363.416,A -85,B 0,C 180,E1 -11443.346,E2 -11443.346} C_VEL
LIN {X 0,Y 395.75,Z 363.74,A -85,B 0,C 180,E1 -11444.394,E2 -11444.394} C_VEL
LIN {X 0,Y 395.805,Z 363.458,A -85,B 0,C 180,E1 -11445.445,E2 -11445.445} C_VEL
LIN {X 0,Y 395.915,Z 362.378,A -85,B 0,C 180,E1 -11446.738,E2 -11446.738} C_VEL
LIN {X 0,Y 396.037,Z 361.345,A -85,B 0,C 180,E1 -11447.557,E2 -11447.557} C_VEL
LIN {X 0,Y 396.301,Z 358.295,A -85,B 0,C 180,E1 -11449.151,E2 -11449.151} C_VEL
LIN {X 0,Y 396.693,Z 353.858,A -85,B 0,C 180,E1 -11450.751,E2 -11450.751} C_VEL
LIN {X 0,Y 396.735,Z 353.141,A -85,B 0,C 180,E1 -11450.948,E2 -11450.948} C_VEL
LIN {X 0,Y 396.293,Z 350.494,A -85,B 0,C 180,E1 -11451.702,E2 -11451.702} C_VEL
LIN {X 0,Y 393.949,Z 345.675,A -85,B 0,C 180,E1 -11452.916,E2 -11452.916} C_VEL
LIN {X 0,Y 391.626,Z 340.204,A -85,B 0,C 180,E1 -11454.074,E2 -11454.074} C_VEL
LIN {X 0,Y 391.22,Z 336.306,A -85,B 0,C 180,E1 -11454.73,E2 -11454.73} C_VEL
LIN {X 0,Y 391.886,Z 329.048,A -85,B 0,C 180,E1 -11455.739,E2 -11455.739} C_VEL
LIN {X 0,Y 392.461,Z 321.561,A -85,B 0,C 180,E1 -11456.594,E2 -11456.594} C_VEL
LIN {X 0,Y 393.072,Z 312.711,A -85,B 0,C 180,E1 -11457.411,E2 -11457.411} C_VEL
LIN {X 0,Y 393.402,Z 306.147,A -85,B 0,C 180,E1 -11457.896,E2 -11457.896} C_VEL
LIN {X 0,Y 391.507,Z 296.071,A -85,B 0,C 180,E1 -11458.603,E2 -11458.603} C_VEL
LIN {X 0,Y 389.068,Z 285.989,A -85,B 0,C 180,E1 -11459.189,E2 -11459.189} C_VEL
LIN {X 0,Y 389.147,Z 282.821,A -85,B 0,C 180,E1 -11461.922,E2 -11461.922} C_VEL
LIN {X 0,Y 389.211,Z 279.027,A -85,B 0,C 180,E1 -11465.296,E2 -11465.296} C_VEL
LIN {X 0,Y 389.352,Z 276.199,A -85,B 0,C 180,E1 -11467.857,E2 -11467.857} C_VEL
LIN {X 0,Y 389.533,Z 273.102,A -85,B 0,C 180,E1 -11470.736,E2 -11470.736} C_VEL
LIN {X 0,Y 389.716,Z 269.82,A -85,B 0,C 180,E1 -11473.838,E2 -11473.838} C_VEL
LIN {X 0,Y 389.722,Z 268.948,A -85,B 0,C 180,E1 -11474.69,E2 -11474.69} C_VEL
LIN {X 0,Y 389.95,Z 268.724,A -85,B 0,C 180,E1 -11477.638,E2 -11477.638} C_VEL
LIN {X 0,Y 390.075,Z 268.71,A -85,B 0,C 180,E1 -11480.909,E2 -11480.909} C_VEL
LIN {X 0,Y 390.066,Z 268.711,A -85,B 0,C 180,E1 -11484.794,E2 -11484.794} C_VEL
LIN {X 0,Y 390.004,Z 268.717,A -85,B 0,C 180,E1 -11488.497,E2 -11488.497} C_VEL
LIN {X 0,Y 390.099,Z 268.707,A -85,B 0,C 180,E1 -11492.071,E2 -11492.071} C_VEL
LIN {X 0,Y 390.06,Z 268.71,A -85,B 0,C 180,E1 -11495.521,E2 -11495.521} C_VEL
LIN {X 0,Y 390.039,Z 268.711,A -85,B 0,C 180,E1 -11498.879,E2 -11498.879} C_VEL
LIN {X 0,Y 390.112,Z 268.7,A -85,B 0,C 180,E1 -11502.168,E2 -11502.168} C_VEL
LIN {X 0,Y 390.132,Z 268.697,A -85,B 0,C 180,E1 -11505.394,E2 -11505.394} C_VEL
LIN {X 0,Y 390.145,Z 268.698,A -85,B 0,C 180,E1 -11508.573,E2 -11508.573} C_VEL
LIN {X 0,Y 390.249,Z 268.686,A -85,B 0,C 180,E1 -11512.081,E2 -11512.081} C_VEL
LIN {X 0,Y 390.207,Z 268.691,A -85,B 0,C 180,E1 -11514.835,E2 -11514.835} C_VEL
LIN {X 0,Y 390.41,Z 268.663,A -85,B 0,C 180,E1 -11517.939,E2 -11517.939} C_VEL
LIN {X 0,Y 390.538,Z 268.65,A -85,B 0,C 180,E1 -11520.002,E2 -11520.002} C_VEL
LIN {X 0,Y 390.3,Z 268.678,A -85,B 0,C 180,E1 -11523.098,E2 -11523.098} C_VEL
LIN {X 0,Y 390.32,Z 268.672,A -85,B 0,C 180,E1 -11526.204,E2 -11526.204} C_VEL
LIN {X 0,Y 390.305,Z 268.681,A -85,B 0,C 180,E1 -11528.284,E2 -11528.284} C_VEL
LIN {X 0,Y 390.168,Z 268.696,A -85,B 0,C 180,E1 -11532.485,E2 -11532.485} C_VEL
LIN {X 0,Y 390.131,Z 268.701,A -85,B 0,C 180,E1 -11535.679,E2 -11535.679} C_VEL
LIN {X 0,Y 390.096,Z 268.705,A -85,B 0,C 180,E1 -11538.924,E2 -11538.924} C_VEL
LIN {X 0,Y 390.03,Z 268.713,A -85,B 0,C 180,E1 -11542.236,E2 -11542.236} C_VEL
LIN {X 0,Y 390.077,Z 268.71,A -85,B 0,C 180,E1 -11545.735,E2 -11545.735} C_VEL
LIN {X 0,Y 390.027,Z 268.72,A -85,B 0,C 180,E1 -11549.114,E2 -11549.114} C_VEL
LIN {X 0,Y 390.037,Z 268.718,A -85,B 0,C 180,E1 -11552.723,E2 -11552.723} C_VEL
LIN {X 0,Y 390.05,Z 268.716,A -85,B 0,C 180,E1 -11555.827,E2 -11555.827} C_VEL
LIN {X 0,Y 390.068,Z 268.711,A -85,B 0,C 180,E1 -11559.221,E2 -11559.221} C_VEL
LIN {X 0,Y 390.076,Z 268.71,A -85,B 0,C 180,E1 -11562.382,E2 -11562.382} C_VEL
LIN {X 0,Y 390.051,Z 268.71,A -85,B 0,C 180,E1 -11566.116,E2 -11566.116} C_VEL
LIN {X 0,Y 390.069,Z 268.77,A -85,B 0,C 180,E1 -11569.721,E2 -11569.721} C_VEL
LIN {X 0,Y 391.011,Z 274.015,A -85,B 0,C 180,E1 -11572.983,E2 -11572.983} C_VEL
LIN {X 0,Y 391.748,Z 278.514,A -85,B 0,C 180,E1 -11575.615,E2 -11575.615} C_VEL
LIN {X 0,Y 391.848,Z 281.902,A -85,B 0,C 180,E1 -11577.456,E2 -11577.456} C_VEL
LIN {X 0,Y 391.128,Z 288.749,A -85,B 0,C 180,E1 -11580.98,E2 -11580.98} C_VEL
LIN {X 0,Y 390.305,Z 296.906,A -85,B 0,C 180,E1 -11584.968,E2 -11584.968} C_VEL
LIN {X 0,Y 389.761,Z 303.97,A -85,B 0,C 180,E1 -11588.308,E2 -11588.308} C_VEL
LIN {X 0,Y 389.343,Z 312.233,A -85,B 0,C 180,E1 -11592.131,E2 -11592.131} C_VEL
LIN {X 0,Y 389.077,Z 318.367,A -85,B 0,C 180,E1 -11594.851,E2 -11594.851} C_VEL
LIN {X 0,Y 391.033,Z 330.612,A -85,B 0,C 180,E1 -11595.428,E2 -11595.428} C_VEL
LIN {X 0,Y 391.956,Z 339.907,A -85,B 0,C 180,E1 -11596.015,E2 -11596.015} C_VEL
LIN {X 0,Y 392.186,Z 348.333,A -85,B 0,C 180,E1 -11596.662,E2 -11596.662} C_VEL
LIN {X 0,Y 391.656,Z 356.716,A -85,B 0,C 180,E1 -11597.435,E2 -11597.435} C_VEL
LIN {X 0,Y 391.065,Z 363.634,A -85,B 0,C 180,E1 -11598.206,E2 -11598.206} C_VEL
LIN {X 0,Y 390.445,Z 370.376,A -85,B 0,C 180,E1 -11599.107,E2 -11599.107} C_VEL
LIN {X 0,Y 389.931,Z 376.782,A -85,B 0,C 180,E1 -11600.142,E2 -11600.142} C_VEL
LIN {X 0,Y 389.482,Z 382.121,A -85,B 0,C 180,E1 -11601.179,E2 -11601.179} C_VEL
LIN {X 0,Y 389.19,Z 386.59,A -85,B 0,C 180,E1 -11602.218,E2 -11602.218} C_VEL
LIN {X 0,Y 388.875,Z 391.701,A -85,B 0,C 180,E1 -11603.724,E2 -11603.724} C_VEL
LIN {X 0,Y 388.793,Z 395.756,A -85,B 0,C 180,E1 -11605.336,E2 -11605.336} C_VEL
LIN {X 0,Y 388.688,Z 398.4,A -85,B 0,C 180,E1 -11606.892,E2 -11606.892} C_VEL
LIN {X 0,Y 388.759,Z 399.431,A -85,B 0,C 180,E1 -11607.929,E2 -11607.929} C_VEL
LIN {X 0,Y 388.761,Z 399.976,A -85,B 0,C 180,E1 -11608.966,E2 -11608.966} C_VEL
LIN {X 0,Y 388.749,Z 400.059,A -85,B 0,C 180,E1 -11610.001,E2 -11610.001} C_VEL
LIN {X 0,Y 388.762,Z 399.677,A -85,B 0,C 180,E1 -11611.037,E2 -11611.037} C_VEL
LIN {X 0,Y 388.798,Z 398.72,A -85,B 0,C 180,E1 -11612.073,E2 -11612.073} C_VEL
LIN {X 0,Y 388.715,Z 396.324,A -85,B 0,C 180,E1 -11613.629,E2 -11613.629} C_VEL
LIN {X 0,Y 388.815,Z 392.585,A -85,B 0,C 180,E1 -11615.187,E2 -11615.187} C_VEL
LIN {X 0,Y 388.877,Z 389.179,A -85,B 0,C 180,E1 -11616.279,E2 -11616.279} C_VEL
LIN {X 0,Y 389.141,Z 384.286,A -85,B 0,C 180,E1 -11617.525,E2 -11617.525} C_VEL
LIN {X 0,Y 389.33,Z 379.309,A -85,B 0,C 180,E1 -11618.566,E2 -11618.566} C_VEL
LIN {X 0,Y 389.62,Z 373.306,A -85,B 0,C 180,E1 -11619.606,E2 -11619.606} C_VEL
LIN {X 0,Y 390.124,Z 366.006,A -85,B 0,C 180,E1 -11620.642,E2 -11620.642} C_VEL
LIN {X 0,Y 390.44,Z 359.422,A -85,B 0,C 180,E1 -11621.421,E2 -11621.421} C_VEL
LIN {X 0,Y 390.973,Z 351.471,A -85,B 0,C 180,E1 -11622.195,E2 -11622.195} C_VEL
LIN {X 0,Y 391.115,Z 344.325,A -85,B 0,C 180,E1 -11622.773,E2 -11622.773} C_VEL
LIN {X 0,Y 390.483,Z 334.763,A -85,B 0,C 180,E1 -11623.398,E2 -11623.398} C_VEL
LIN {X 0,Y 389.575,Z 325.425,A -85,B 0,C 180,E1 -11623.864,E2 -11623.864} C_VEL
LIN {X 0,Y 388.899,Z 318.641,A -85,B 0,C 180,E1 -11624.122,E2 -11624.122} C_VEL
LIN {X 0,Y 389.139,Z 311.46,A -85,B 0,C 180,E1 -11627.284,E2 -11627.284} C_VEL
LIN {X 0,Y 389.455,Z 303.987,A -85,B 0,C 180,E1 -11630.617,E2 -11630.617} C_VEL
LIN {X 0,Y 389.882,Z 296.652,A -85,B 0,C 180,E1 -11633.929,E2 -11633.929} C_VEL
LIN {X 0,Y 390.409,Z 289.303,A -85,B 0,C 180,E1 -11637.327,E2 -11637.327} C_VEL
LIN {X 0,Y 391.055,Z 281.895,A -85,B 0,C 180,E1 -11640.83,E2 -11640.83} C_VEL
LIN {X 0,Y 391.402,Z 277.015,A -85,B 0,C 180,E1 -11643.208,E2 -11643.208} C_VEL
LIN {X 0,Y 390.616,Z 271.778,A -85,B 0,C 180,E1 -11645.937,E2 -11645.937} C_VEL
LIN {X 0,Y 390.091,Z 268.708,A -85,B 0,C 180,E1 -11647.626,E2 -11647.626} C_VEL
LIN {X 0,Y 390.065,Z 268.708,A -85,B 0,C 180,E1 -11650.821,E2 -11650.821} C_VEL
LIN {X 0,Y 390.064,Z 268.712,A -85,B 0,C 180,E1 -11653.886,E2 -11653.886} C_VEL
LIN {X 0,Y 390.066,Z 268.707,A -85,B 0,C 180,E1 -11656.789,E2 -11656.789} C_VEL
LIN {X 0,Y 390.066,Z 268.711,A -85,B 0,C 180,E1 -11659.56,E2 -11659.56} C_VEL
LIN {X 0,Y 390.051,Z 268.71,A -85,B 0,C 180,E1 -11662.449,E2 -11662.449} C_VEL
LIN {X 0,Y 390.078,Z 268.709,A -85,B 0,C 180,E1 -11665.975,E2 -11665.975} C_VEL
LIN {X 0,Y 390.056,Z 268.712,A -85,B 0,C 180,E1 -11669.868,E2 -11669.868} C_VEL
LIN {X 0,Y 390.123,Z 268.704,A -85,B 0,C 180,E1 -11673.231,E2 -11673.231} C_VEL
LIN {X 0,Y 390.086,Z 268.707,A -85,B 0,C 180,E1 -11676.76,E2 -11676.76} C_VEL
LIN {X 0,Y 390.113,Z 268.702,A -85,B 0,C 180,E1 -11679.982,E2 -11679.982} C_VEL
LIN {X 0,Y 390.147,Z 268.702,A -85,B 0,C 180,E1 -11683.247,E2 -11683.247} C_VEL
LIN {X 0,Y 390.203,Z 268.693,A -85,B 0,C 180,E1 -11686.56,E2 -11686.56} C_VEL
LIN {X 0,Y 390.175,Z 268.695,A -85,B 0,C 180,E1 -11689.621,E2 -11689.621} C_VEL
LIN {X 0,Y 390.289,Z 268.684,A -85,B 0,C 180,E1 -11692.757,E2 -11692.757} C_VEL
LIN {X 0,Y 390.229,Z 268.692,A -85,B 0,C 180,E1 -11694.832,E2 -11694.832} C_VEL
LIN {X 0,Y 390.424,Z 268.664,A -85,B 0,C 180,E1 -11697.935,E2 -11697.935} C_VEL
LIN {X 0,Y 390.554,Z 268.648,A -85,B 0,C 180,E1 -11699.998,E2 -11699.998} C_VEL
LIN {X 0,Y 390.32,Z 268.677,A -85,B 0,C 180,E1 -11703.095,E2 -11703.095} C_VEL
LIN {X 0,Y 390.315,Z 268.677,A -85,B 0,C 180,E1 -11706.617,E2 -11706.617} C_VEL
LIN {X 0,Y 390.209,Z 268.69,A -85,B 0,C 180,E1 -11709.327,E2 -11709.327} C_VEL
LIN {X 0,Y 390.197,Z 268.692,A -85,B 0,C 180,E1 -11713.436,E2 -11713.436} C_VEL
LIN {X 0,Y 390.15,Z 268.698,A -85,B 0,C 180,E1 -11717.305,E2 -11717.305} C_VEL
LIN {X 0,Y 390.088,Z 268.707,A -85,B 0,C 180,E1 -11720.468,E2 -11720.468} C_VEL
LIN {X 0,Y 390.089,Z 268.706,A -85,B 0,C 180,E1 -11723.348,E2 -11723.348} C_VEL
LIN {X 0,Y 390.112,Z 268.702,A -85,B 0,C 180,E1 -11726.766,E2 -11726.766} C_VEL
LIN {X 0,Y 390.036,Z 268.712,A -85,B 0,C 180,E1 -11730.297,E2 -11730.297} C_VEL
LIN {X 0,Y 390.064,Z 268.71,A -85,B 0,C 180,E1 -11734.022,E2 -11734.022} C_VEL
LIN {X 0,Y 390.042,Z 268.715,A -85,B 0,C 180,E1 -11737.549,E2 -11737.549} C_VEL
LIN {X 0,Y 390.076,Z 268.708,A -85,B 0,C 180,E1 -11740.823,E2 -11740.823} C_VEL
LIN {X 0,Y 390.122,Z 268.702,A -85,B 0,C 180,E1 -11743.895,E2 -11743.895} C_VEL
LIN {X 0,Y 390.112,Z 268.704,A -85,B 0,C 180,E1 -11747.611,E2 -11747.611} C_VEL
LIN {X 0,Y 390.085,Z 268.709,A -85,B 0,C 180,E1 -11750.906,E2 -11750.906} C_VEL
LIN {X 0,Y 390.074,Z 268.711,A -85,B 0,C 180,E1 -11754.791,E2 -11754.791} C_VEL
LIN {X 0,Y 390.015,Z 268.716,A -85,B 0,C 180,E1 -11758.494,E2 -11758.494} C_VEL
LIN {X 0,Y 390.104,Z 268.704,A -85,B 0,C 180,E1 -11762.068,E2 -11762.068} C_VEL
LIN {X 0,Y 390.067,Z 268.708,A -85,B 0,C 180,E1 -11765.517,E2 -11765.517} C_VEL
LIN {X 0,Y 390.063,Z 268.711,A -85,B 0,C 180,E1 -11768.877,E2 -11768.877} C_VEL
LIN {X 0,Y 390.004,Z 268.717,A -85,B 0,C 180,E1 -11771.072,E2 -11771.072} C_VEL
LIN {X 0,Y 389.83,Z 268.738,A -85,B 0,C 180,E1 -11773.233,E2 -11773.233} C_VEL
LIN {X 0,Y 389.517,Z 268.78,A -85,B 0,C 180,E1 -11775.367,E2 -11775.367} C_VEL
LIN {X 0,Y 389.518,Z 270.131,A -85,B 0,C 180,E1 -11776.971,E2 -11776.971} C_VEL
LIN {X 0,Y 389.346,Z 274.415,A -85,B 0,C 180,E1 -11780.649,E2 -11780.649} C_VEL
LIN {X 0,Y 389.345,Z 278.071,A -85,B 0,C 180,E1 -11783.781,E2 -11783.781} C_VEL
LIN {X 0,Y 389.229,Z 281.795,A -85,B 0,C 180,E1 -11786.894,E2 -11786.894} C_VEL
LIN {X 0,Y 388.997,Z 285.591,A -85,B 0,C 180,E1 -11789.999,E2 -11789.999} C_VEL
LIN {X 0,Y 390.92,Z 297.247,A -85,B 0,C 180,E1 -11790.578,E2 -11790.578} C_VEL
LIN {X 0,Y 391.901,Z 304.436,A -85,B 0,C 180,E1 -11791.026,E2 -11791.026} C_VEL
LIN {X 0,Y 391.553,Z 313.176,A -85,B 0,C 180,E1 -11791.67,E2 -11791.67} C_VEL
LIN {X 0,Y 391.124,Z 321.534,A -85,B 0,C 180,E1 -11792.445,E2 -11792.445} C_VEL
LIN {X 0,Y 390.634,Z 329.451,A -85,B 0,C 180,E1 -11793.351,E2 -11793.351} C_VEL
LIN {X 0,Y 390.235,Z 336.821,A -85,B 0,C 180,E1 -11794.388,E2 -11794.388} C_VEL
LIN {X 0,Y 389.744,Z 344.313,A -85,B 0,C 180,E1 -11795.69,E2 -11795.69} C_VEL
LIN {X 0,Y 389.499,Z 350.523,A -85,B 0,C 180,E1 -11797.091,E2 -11797.091} C_VEL
LIN {X 0,Y 389.178,Z 354.799,A -85,B 0,C 180,E1 -11798.305,E2 -11798.305} C_VEL
LIN {X 0,Y 388.993,Z 357.804,A -85,B 0,C 180,E1 -11799.357,E2 -11799.357} C_VEL
LIN {X 0,Y 388.838,Z 360.151,A -85,B 0,C 180,E1 -11800.412,E2 -11800.412} C_VEL
LIN {X 0,Y 388.772,Z 361.878,A -85,B 0,C 180,E1 -11801.468,E2 -11801.468} C_VEL
LIN {X 0,Y 388.717,Z 363.093,A -85,B 0,C 180,E1 -11802.529,E2 -11802.529} C_VEL
LIN {X 0,Y 388.666,Z 363.814,A -85,B 0,C 180,E1 -11803.594,E2 -11803.594} C_VEL
LIN {X 0,Y 388.662,Z 364.044,A -85,B 0,C 180,E1 -11804.663,E2 -11804.663} C_VEL
LIN {X 0,Y 388.76,Z 363.721,A -85,B 0,C 180,E1 -11805.732,E2 -11805.732} C_VEL
LIN {X 0,Y 388.858,Z 362.802,A -85,B 0,C 180,E1 -11806.807,E2 -11806.807} C_VEL
LIN {X 0,Y 389.09,Z 360.506,A -85,B 0,C 180,E1 -11808.425,E2 -11808.425} C_VEL
LIN {X 0,Y 389.46,Z 356.745,A -85,B 0,C 180,E1 -11810.05,E2 -11810.05} C_VEL
LIN {X 0,Y 389.739,Z 353.458,A -85,B 0,C 180,E1 -11811.139,E2 -11811.139} C_VEL
LIN {X 0,Y 390.198,Z 348.182,A -85,B 0,C 180,E1 -11812.502,E2 -11812.502} C_VEL
LIN {X 0,Y 390.697,Z 343.114,A -85,B 0,C 180,E1 -11813.563,E2 -11813.563} C_VEL
LIN {X 0,Y 391.22,Z 336.306,A -85,B 0,C 180,E1 -11814.73,E2 -11814.73} C_VEL
LIN {X 0,Y 390.829,Z 332.335,A -85,B 0,C 180,E1 -11815.353,E2 -11815.353} C_VEL
LIN {X 0,Y 388.634,Z 325.437,A -85,B 0,C 180,E1 -11816.343,E2 -11816.343} C_VEL
LIN {X 0,Y 386.537,Z 317.963,A -85,B 0,C 180,E1 -11817.247,E2 -11817.247} C_VEL
LIN {X 0,Y 386.316,Z 312.848,A -85,B 0,C 180,E1 -11817.725,E2 -11817.725} C_VEL
LIN {X 0,Y 386.585,Z 307.471,A -85,B 0,C 180,E1 -11818.132,E2 -11818.132} C_VEL
LIN {X 0,Y 384.944,Z 298.417,A -85,B 0,C 180,E1 -11818.801,E2 -11818.801} C_VEL
LIN {X 0,Y 382.433,Z 288.27,A -85,B 0,C 180,E1 -11819.412,E2 -11819.412} C_VEL
LIN {X 0,Y 382.025,Z 286.301,A -85,B 0,C 180,E1 -11819.55,E2 -11819.55} C_VEL
LIN {X 0,Y 382.102,Z 283.245,A -85,B 0,C 180,E1 -11822.233,E2 -11822.233} C_VEL
LIN {X 0,Y 382.212,Z 279.057,A -85,B 0,C 180,E1 -11826.042,E2 -11826.042} C_VEL
LIN {X 0,Y 382.389,Z 275.341,A -85,B 0,C 180,E1 -11829.477,E2 -11829.477} C_VEL
LIN {X 0,Y 382.585,Z 271.849,A -85,B 0,C 180,E1 -11832.816,E2 -11832.816} C_VEL
LIN {X 0,Y 382.694,Z 270.352,A -85,B 0,C 180,E1 -11834.261,E2 -11834.261} C_VEL
LIN {X 0,Y 382.793,Z 269.614,A -85,B 0,C 180,E1 -11835.763,E2 -11835.763} C_VEL
LIN {X 0,Y 382.941,Z 269.597,A -85,B 0,C 180,E1 -11838.801,E2 -11838.801} C_VEL
LIN {X 0,Y 382.984,Z 269.594,A -85,B 0,C 180,E1 -11842.096,E2 -11842.096} C_VEL
LIN {X 0,Y 382.999,Z 269.591,A -85,B 0,C 180,E1 -11845.333,E2 -11845.333} C_VEL
LIN {X 0,Y 382.964,Z 269.595,A -85,B 0,C 180,E1 -11849.083,E2 -11849.083} C_VEL
LIN {X 0,Y 383.039,Z 269.585,A -85,B 0,C 180,E1 -11852.699,E2 -11852.699} C_VEL
LIN {X 0,Y 383.033,Z 269.587,A -85,B 0,C 180,E1 -11855.041,E2 -11855.041} C_VEL
LIN {X 0,Y 382.975,Z 269.593,A -85,B 0,C 180,E1 -11858.47,E2 -11858.47} C_VEL
LIN {X 0,Y 383.073,Z 269.579,A -85,B 0,C 180,E1 -11861.829,E2 -11861.829} C_VEL
LIN {X 0,Y 383.097,Z 269.575,A -85,B 0,C 180,E1 -11865.12,E2 -11865.12} C_VEL
LIN {X 0,Y 383.094,Z 269.577,A -85,B 0,C 180,E1 -11868.36,E2 -11868.36} C_VEL
LIN {X 0,Y 383.208,Z 269.563,A -85,B 0,C 180,E1 -11872.022,E2 -11872.022} C_VEL
LIN {X 0,Y 383.177,Z 269.567,A -85,B 0,C 180,E1 -11874.74,E2 -11874.74} C_VEL
LIN {X 0,Y 383.377,Z 269.539,A -85,B 0,C 180,E1 -11877.901,E2 -11877.901} C_VEL
LIN {X 0,Y 383.507,Z 269.526,A -85,B 0,C 180,E1 -11880.002,E2 -11880.002} C_VEL
LIN {X 0,Y 383.236,Z 269.558,A -85,B 0,C 180,E1 -11883.156,E2 -11883.156} C_VEL
LIN {X 0,Y 383.278,Z 269.55,A -85,B 0,C 180,E1 -11886.318,E2 -11886.318} C_VEL
LIN {X 0,Y 383.25,Z 269.561,A -85,B 0,C 180,E1 -11888.438,E2 -11888.438} C_VEL
LIN {X 0,Y 383.096,Z 269.579,A -85,B 0,C 180,E1 -11891.644,E2 -11891.644} C_VEL
LIN {X 0,Y 383.103,Z 269.579,A -85,B 0,C 180,E1 -11894.884,E2 -11894.884} C_VEL
LIN {X 0,Y 383.08,Z 269.581,A -85,B 0,C 180,E1 -11898.174,E2 -11898.174} C_VEL
LIN {X 0,Y 382.984,Z 269.593,A -85,B 0,C 180,E1 -11901.533,E2 -11901.533} C_VEL
LIN {X 0,Y 383.022,Z 269.588,A -85,B 0,C 180,E1 -11904.964,E2 -11904.964} C_VEL
LIN {X 0,Y 382.979,Z 269.594,A -85,B 0,C 180,E1 -11908.499,E2 -11908.499} C_VEL
LIN {X 0,Y 383.004,Z 269.595,A -85,B 0,C 180,E1 -11912.152,E2 -11912.152} C_VEL
LIN {X 0,Y 383.013,Z 269.592,A -85,B 0,C 180,E1 -11914.67,E2 -11914.67} C_VEL
LIN {X 0,Y 382.997,Z 269.591,A -85,B 0,C 180,E1 -11917.906,E2 -11917.906} C_VEL
LIN {X 0,Y 383.009,Z 269.589,A -85,B 0,C 180,E1 -11921.346,E2 -11921.346} C_VEL
LIN {X 0,Y 382.993,Z 269.595,A -85,B 0,C 180,E1 -11924.305,E2 -11924.305} C_VEL
LIN {X 0,Y 383.007,Z 269.595,A -85,B 0,C 180,E1 -11927.242,E2 -11927.242} C_VEL
LIN {X 0,Y 383.037,Z 269.681,A -85,B 0,C 180,E1 -11929.358,E2 -11929.358} C_VEL
LIN {X 0,Y 384.008,Z 275.134,A -85,B 0,C 180,E1 -11932.848,E2 -11932.848} C_VEL
LIN {X 0,Y 384.85,Z 280.723,A -85,B 0,C 180,E1 -11936.155,E2 -11936.155} C_VEL
LIN {X 0,Y 384.711,Z 284.135,A -85,B 0,C 180,E1 -11938.011,E2 -11938.011} C_VEL
LIN {X 0,Y 384.086,Z 289.849,A -85,B 0,C 180,E1 -11940.997,E2 -11940.997} C_VEL
LIN {X 0,Y 383.249,Z 297.978,A -85,B 0,C 180,E1 -11945.055,E2 -11945.055} C_VEL
LIN {X 0,Y 382.679,Z 304.992,A -85,B 0,C 180,E1 -11948.452,E2 -11948.452} C_VEL
LIN {X 0,Y 382.255,Z 313.25,A -85,B 0,C 180,E1 -11952.342,E2 -11952.342} C_VEL
LIN {X 0,Y 382.019,Z 317.937,A -85,B 0,C 180,E1 -11954.496,E2 -11954.496} C_VEL
LIN {X 0,Y 384.015,Z 330.162,A -85,B 0,C 180,E1 -11955.088,E2 -11955.088} C_VEL
LIN {X 0,Y 385.078,Z 340.529,A -85,B 0,C 180,E1 -11955.772,E2 -11955.772} C_VEL
LIN {X 0,Y 385.28,Z 348.637,A -85,B 0,C 180,E1 -11956.418,E2 -11956.418} C_VEL
LIN {X 0,Y 384.735,Z 356.905,A -85,B 0,C 180,E1 -11957.205,E2 -11957.205} C_VEL
LIN {X 0,Y 384.112,Z 363.735,A -85,B 0,C 180,E1 -11957.989,E2 -11957.989} C_VEL
LIN {X 0,Y 383.482,Z 370.405,A -85,B 0,C 180,E1 -11958.907,E2 -11958.907} C_VEL
LIN {X 0,Y 382.922,Z 376.75,A -85,B 0,C 180,E1 -11959.96,E2 -11959.96} C_VEL
LIN {X 0,Y 382.462,Z 382.037,A -85,B 0,C 180,E1 -11961.015,E2 -11961.015} C_VEL
LIN {X 0,Y 382.133,Z 386.46,A -85,B 0,C 180,E1 -11962.073,E2 -11962.073} C_VEL
LIN {X 0,Y 381.811,Z 391.685,A -85,B 0,C 180,E1 -11963.661,E2 -11963.661} C_VEL
LIN {X 0,Y 381.697,Z 394.379,A -85,B 0,C 180,E1 -11964.719,E2 -11964.719} C_VEL
LIN {X 0,Y 381.676,Z 396.525,A -85,B 0,C 180,E1 -11965.778,E2 -11965.778} C_VEL
LIN {X 0,Y 381.597,Z 398.137,A -85,B 0,C 180,E1 -11966.834,E2 -11966.834} C_VEL
LIN {X 0,Y 381.657,Z 399.149,A -85,B 0,C 180,E1 -11967.891,E2 -11967.891} C_VEL
LIN {X 0,Y 381.692,Z 399.662,A -85,B 0,C 180,E1 -11968.946,E2 -11968.946} C_VEL
LIN {X 0,Y 381.678,Z 399.713,A -85,B 0,C 180,E1 -11970.001,E2 -11970.001} C_VEL
LIN {X 0,Y 381.694,Z 399.301,A -85,B 0,C 180,E1 -11971.056,E2 -11971.056} C_VEL
LIN {X 0,Y 381.699,Z 398.338,A -85,B 0,C 180,E1 -11972.112,E2 -11972.112} C_VEL
LIN {X 0,Y 381.633,Z 395.881,A -85,B 0,C 180,E1 -11973.697,E2 -11973.697} C_VEL
LIN {X 0,Y 381.723,Z 393.559,A -85,B 0,C 180,E1 -11974.754,E2 -11974.754} C_VEL
LIN {X 0,Y 381.813,Z 388.844,A -85,B 0,C 180,E1 -11976.342,E2 -11976.342} C_VEL
LIN {X 0,Y 382.052,Z 383.704,A -85,B 0,C 180,E1 -11977.665,E2 -11977.665} C_VEL
LIN {X 0,Y 382.276,Z 378.674,A -85,B 0,C 180,E1 -11978.725,E2 -11978.725} C_VEL
LIN {X 0,Y 382.608,Z 372.61,A -85,B 0,C 180,E1 -11979.784,E2 -11979.784} C_VEL
LIN {X 0,Y 383.057,Z 365.228,A -85,B 0,C 180,E1 -11980.841,E2 -11980.841} C_VEL
LIN {X 0,Y 383.533,Z 357.322,A -85,B 0,C 180,E1 -11981.764,E2 -11981.764} C_VEL
LIN {X 0,Y 384.06,Z 348.98,A -85,B 0,C 180,E1 -11982.552,E2 -11982.552} C_VEL
LIN {X 0,Y 383.946,Z 342.291,A -85,B 0,C 180,E1 -11983.076,E2 -11983.076} C_VEL
LIN {X 0,Y 383.298,Z 333.605,A -85,B 0,C 180,E1 -11983.639,E2 -11983.639} C_VEL
LIN {X 0,Y 382.394,Z 324.02,A -85,B 0,C 180,E1 -11984.113,E2 -11984.113} C_VEL
LIN {X 0,Y 381.838,Z 318.278,A -85,B 0,C 180,E1 -11984.355,E2 -11984.355} C_VEL
LIN {X 0,Y 382.074,Z 310.925,A -85,B 0,C 180,E1 -11987.67,E2 -11987.67} C_VEL
LIN {X 0,Y 382.484,Z 302.384,A -85,B 0,C 180,E1 -11991.562,E2 -11991.562} C_VEL
LIN {X 0,Y 382.943,Z 295.046,A -85,B 0,C 180,E1 -11994.969,E2 -11994.969} C_VEL
LIN {X 0,Y 383.517,Z 287.819,A -85,B 0,C 180,E1 -11998.403,E2 -11998.403} C_VEL
LIN {X 0,Y 384.074,Z 281.573,A -85,B 0,C 180,E1 -12001.435,E2 -12001.435} C_VEL
LIN {X 0,Y 384.365,Z 277.913,A -85,B 0,C 180,E1 -12003.268,E2 -12003.268} C_VEL
LIN {X 0,Y 383.642,Z 272.958,A -85,B 0,C 180,E1 -12005.89,E2 -12005.89} C_VEL
LIN {X 0,Y 383.076,Z 269.582,A -85,B 0,C 180,E1 -12007.823,E2 -12007.823} C_VEL
LIN {X 0,Y 382.992,Z 269.589,A -85,B 0,C 180,E1 -12011.348,E2 -12011.348} C_VEL
LIN {X 0,Y 383.005,Z 269.59,A -85,B 0,C 180,E1 -12014.303,E2 -12014.303} C_VEL
LIN {X 0,Y 383.02,Z 269.586,A -85,B 0,C 180,E1 -12017.24,E2 -12017.24} C_VEL
LIN {X 0,Y 383.022,Z 269.586,A -85,B 0,C 180,E1 -12020.414,E2 -12020.414} C_VEL
LIN {X 0,Y 383.034,Z 269.586,A -85,B 0,C 180,E1 -12024.044,E2 -12024.044} C_VEL
LIN {X 0,Y 382.996,Z 269.593,A -85,B 0,C 180,E1 -12027.578,E2 -12027.578} C_VEL
LIN {X 0,Y 383.001,Z 269.588,A -85,B 0,C 180,E1 -12030.299,E2 -12030.299} C_VEL
LIN {X 0,Y 383.066,Z 269.58,A -85,B 0,C 180,E1 -12032.697,E2 -12032.697} C_VEL
LIN {X 0,Y 383.06,Z 269.583,A -85,B 0,C 180,E1 -12035.039,E2 -12035.039} C_VEL
LIN {X 0,Y 383.001,Z 269.588,A -85,B 0,C 180,E1 -12038.468,E2 -12038.468} C_VEL
LIN {X 0,Y 383.062,Z 269.581,A -85,B 0,C 180,E1 -12041.825,E2 -12041.825} C_VEL
LIN {X 0,Y 383.119,Z 269.577,A -85,B 0,C 180,E1 -12045.117,E2 -12045.117} C_VEL
LIN {X 0,Y 383.104,Z 269.576,A -85,B 0,C 180,E1 -12048.356,E2 -12048.356} C_VEL
LIN {X 0,Y 383.235,Z 269.559,A -85,B 0,C 180,E1 -12052.013,E2 -12052.013} C_VEL
LIN {X 0,Y 383.201,Z 269.567,A -85,B 0,C 180,E1 -12054.737,E2 -12054.737} C_VEL
LIN {X 0,Y 383.392,Z 269.539,A -85,B 0,C 180,E1 -12057.897,E2 -12057.897} C_VEL
LIN {X 0,Y 383.524,Z 269.523,A -85,B 0,C 180,E1 -12059.998,E2 -12059.998} C_VEL
LIN {X 0,Y 383.256,Z 269.556,A -85,B 0,C 180,E1 -12063.152,E2 -12063.152} C_VEL
LIN {X 0,Y 383.275,Z 269.555,A -85,B 0,C 180,E1 -12066.611,E2 -12066.611} C_VEL
LIN {X 0,Y 383.265,Z 269.559,A -85,B 0,C 180,E1 -12068.434,E2 -12068.434} C_VEL
LIN {X 0,Y 383.101,Z 269.576,A -85,B 0,C 180,E1 -12071.64,E2 -12071.64} C_VEL
LIN {X 0,Y 383.112,Z 269.574,A -85,B 0,C 180,E1 -12074.879,E2 -12074.879} C_VEL
LIN {X 0,Y 383.091,Z 269.581,A -85,B 0,C 180,E1 -12078.17,E2 -12078.17} C_VEL
LIN {X 0,Y 382.993,Z 269.591,A -85,B 0,C 180,E1 -12081.528,E2 -12081.528} C_VEL
LIN {X 0,Y 383.051,Z 269.581,A -85,B 0,C 180,E1 -12084.958,E2 -12084.958} C_VEL
LIN {X 0,Y 383.028,Z 269.586,A -85,B 0,C 180,E1 -12088.268,E2 -12088.268} C_VEL
LIN {X 0,Y 383.006,Z 269.589,A -85,B 0,C 180,E1 -12092.147,E2 -12092.147} C_VEL
LIN {X 0,Y 383.014,Z 269.586,A -85,B 0,C 180,E1 -12094.665,E2 -12094.665} C_VEL
LIN {X 0,Y 382.998,Z 269.59,A -85,B 0,C 180,E1 -12097.902,E2 -12097.902} C_VEL
LIN {X 0,Y 383.04,Z 269.587,A -85,B 0,C 180,E1 -12101.336,E2 -12101.336} C_VEL
LIN {X 0,Y 383.063,Z 269.58,A -85,B 0,C 180,E1 -12104.312,E2 -12104.312} C_VEL
LIN {X 0,Y 383.067,Z 269.584,A -85,B 0,C 180,E1 -12107.247,E2 -12107.247} C_VEL
LIN {X 0,Y 383.013,Z 269.587,A -85,B 0,C 180,E1 -12110.41,E2 -12110.41} C_VEL
LIN {X 0,Y 383.016,Z 269.585,A -85,B 0,C 180,E1 -12114.042,E2 -12114.042} C_VEL
LIN {X 0,Y 382.976,Z 269.591,A -85,B 0,C 180,E1 -12117.575,E2 -12117.575} C_VEL
LIN {X 0,Y 382.985,Z 269.591,A -85,B 0,C 180,E1 -12120.298,E2 -12120.298} C_VEL
LIN {X 0,Y 383.043,Z 269.587,A -85,B 0,C 180,E1 -12122.696,E2 -12122.696} C_VEL
LIN {X 0,Y 383.028,Z 269.586,A -85,B 0,C 180,E1 -12126.191,E2 -12126.191} C_VEL
LIN {X 0,Y 383.046,Z 269.582,A -85,B 0,C 180,E1 -12129.597,E2 -12129.597} C_VEL
LIN {X 0,Y 382.821,Z 269.612,A -85,B 0,C 180,E1 -12132.917,E2 -12132.917} C_VEL
LIN {X 0,Y 382.508,Z 269.653,A -85,B 0,C 180,E1 -12135.093,E2 -12135.093} C_VEL
LIN {X 0,Y 382.416,Z 269.987,A -85,B 0,C 180,E1 -12136.176,E2 -12136.176} C_VEL
LIN {X 0,Y 382.371,Z 272.427,A -85,B 0,C 180,E1 -12138.334,E2 -12138.334} C_VEL
LIN {X 0,Y 382.31,Z 277.327,A -85,B 0,C 180,E1 -12142.605,E2 -12142.605} C_VEL
LIN {X 0,Y 382.255,Z 281.055,A -85,B 0,C 180,E1 -12145.781,E2 -12145.781} C_VEL
LIN {X 0,Y 382.01,Z 284.865,A -85,B 0,C 180,E1 -12148.944,E2 -12148.944} C_VEL
LIN {X 0,Y 381.939,Z 285.905,A -85,B 0,C 180,E1 -12149.801,E2 -12149.801} C_VEL
LIN {X 0,Y 383.86,Z 297.727,A -85,B 0,C 180,E1 -12150.392,E2 -12150.392} C_VEL
LIN {X 0,Y 384.862,Z 303.952,A -85,B 0,C 180,E1 -12150.783,E2 -12150.783} C_VEL
LIN {X 0,Y 384.607,Z 312.813,A -85,B 0,C 180,E1 -12151.438,E2 -12151.438} C_VEL
LIN {X 0,Y 384.147,Z 321.298,A -85,B 0,C 180,E1 -12152.227,E2 -12152.227} C_VEL
LIN {X 0,Y 383.629,Z 329.312,A -85,B 0,C 180,E1 -12153.149,E2 -12153.149} C_VEL
LIN {X 0,Y 383.318,Z 335.052,A -85,B 0,C 180,E1 -12153.941,E2 -12153.941} C_VEL
LIN {X 0,Y 382.91,Z 341.466,A -85,B 0,C 180,E1 -12155,E2 -12155} C_VEL
LIN {X 0,Y 382.632,Z 346.789,A -85,B 0,C 180,E1 -12156.061,E2 -12156.061} C_VEL
LIN {X 0,Y 382.406,Z 351.068,A -85,B 0,C 180,E1 -12157.078,E2 -12157.078} C_VEL
LIN {X 0,Y 382.069,Z 355.719,A -85,B 0,C 180,E1 -12158.461,E2 -12158.461} C_VEL
LIN {X 0,Y 381.79,Z 359.761,A -85,B 0,C 180,E1 -12160.07,E2 -12160.07} C_VEL
LIN {X 0,Y 381.662,Z 362.529,A -85,B 0,C 180,E1 -12161.685,E2 -12161.685} C_VEL
LIN {X 0,Y 381.628,Z 363.615,A -85,B 0,C 180,E1 -12162.766,E2 -12162.766} C_VEL
LIN {X 0,Y 381.565,Z 364.211,A -85,B 0,C 180,E1 -12163.852,E2 -12163.852} C_VEL
LIN {X 0,Y 381.584,Z 364.315,A -85,B 0,C 180,E1 -12164.941,E2 -12164.941} C_VEL
LIN {X 0,Y 381.683,Z 363.92,A -85,B 0,C 180,E1 -12166.032,E2 -12166.032} C_VEL
LIN {X 0,Y 381.808,Z 362.945,A -85,B 0,C 180,E1 -12167.127,E2 -12167.127} C_VEL
LIN {X 0,Y 382.078,Z 360.411,A -85,B 0,C 180,E1 -12168.776,E2 -12168.776} C_VEL
LIN {X 0,Y 382.361,Z 358.013,A -85,B 0,C 180,E1 -12169.878,E2 -12169.878} C_VEL
LIN {X 0,Y 382.796,Z 353.024,A -85,B 0,C 180,E1 -12171.541,E2 -12171.541} C_VEL
LIN {X 0,Y 383.197,Z 348.789,A -85,B 0,C 180,E1 -12172.651,E2 -12172.651} C_VEL
LIN {X 0,Y 383.752,Z 343.633,A -85,B 0,C 180,E1 -12173.758,E2 -12173.758} C_VEL
LIN {X 0,Y 384.267,Z 337.15,A -85,B 0,C 180,E1 -12174.902,E2 -12174.902} C_VEL
LIN {X 0,Y 384.905,Z 330.648,A -85,B 0,C 180,E1 -12175.843,E2 -12175.843} C_VEL
LIN {X 0,Y 385.502,Z 323.41,A -85,B 0,C 180,E1 -12176.715,E2 -12176.715} C_VEL
LIN {X 0,Y 386.137,Z 315.358,A -85,B 0,C 180,E1 -12177.504,E2 -12177.504} C_VEL
LIN {X 0,Y 386.316,Z 312.848,A -85,B 0,C 180,E1 -12177.725,E2 -12177.725} C_VEL
LIN {X 0,Y 385.755,Z 309.585,A -85,B 0,C 180,E1 -12178.033,E2 -12178.033} C_VEL
LIN {X 0,Y 384.071,Z 306.621,A -85,B 0,C 180,E1 -12178.343,E2 -12178.343} C_VEL
LIN {X 0,Y 378.906,Z 299.949,A -85,B 0,C 180,E1 -12179.029,E2 -12179.029} C_VEL
LIN {X 0,Y 377.449,Z 296.583,A -85,B 0,C 180,E1 -12179.303,E2 -12179.303} C_VEL
LIN {X 0,Y 374.943,Z 286.639,A -85,B 0,C 180,E1 -12179.915,E2 -12179.915} C_VEL
LIN {X 0,Y 375.023,Z 283.285,A -85,B 0,C 180,E1 -12182.918,E2 -12182.918} C_VEL
LIN {X 0,Y 375.175,Z 279.563,A -85,B 0,C 180,E1 -12186.346,E2 -12186.346} C_VEL
LIN {X 0,Y 375.377,Z 275.832,A -85,B 0,C 180,E1 -12189.864,E2 -12189.864} C_VEL
LIN {X 0,Y 375.551,Z 272.476,A -85,B 0,C 180,E1 -12193.131,E2 -12193.131} C_VEL
LIN {X 0,Y 375.668,Z 270.502,A -85,B 0,C 180,E1 -12195.306,E2 -12195.306} C_VEL
LIN {X 0,Y 375.871,Z 270.479,A -85,B 0,C 180,E1 -12198.407,E2 -12198.407} C_VEL
LIN {X 0,Y 375.958,Z 270.469,A -85,B 0,C 180,E1 -12201.73,E2 -12201.73} C_VEL
LIN {X 0,Y 375.961,Z 270.468,A -85,B 0,C 180,E1 -12205.334,E2 -12205.334} C_VEL
LIN {X 0,Y 375.939,Z 270.469,A -85,B 0,C 180,E1 -12208.439,E2 -12208.439} C_VEL
LIN {X 0,Y 375.965,Z 270.468,A -85,B 0,C 180,E1 -12212.142,E2 -12212.142} C_VEL
LIN {X 0,Y 375.988,Z 270.463,A -85,B 0,C 180,E1 -12214.54,E2 -12214.54} C_VEL
LIN {X 0,Y 375.941,Z 270.469,A -85,B 0,C 180,E1 -12218.047,E2 -12218.047} C_VEL
LIN {X 0,Y 376.008,Z 270.462,A -85,B 0,C 180,E1 -12221.476,E2 -12221.476} C_VEL
LIN {X 0,Y 376.044,Z 270.456,A -85,B 0,C 180,E1 -12224.834,E2 -12224.834} C_VEL
LIN {X 0,Y 376.045,Z 270.457,A -85,B 0,C 180,E1 -12228.139,E2 -12228.139} C_VEL
LIN {X 0,Y 376.18,Z 270.438,A -85,B 0,C 180,E1 -12231.948,E2 -12231.948} C_VEL
LIN {X 0,Y 376.148,Z 270.444,A -85,B 0,C 180,E1 -12234.642,E2 -12234.642} C_VEL
LIN {X 0,Y 376.343,Z 270.415,A -85,B 0,C 180,E1 -12237.862,E2 -12237.862} C_VEL
LIN {X 0,Y 376.477,Z 270.402,A -85,B 0,C 180,E1 -12240.002,E2 -12240.002} C_VEL
LIN {X 0,Y 376.175,Z 270.438,A -85,B 0,C 180,E1 -12243.215,E2 -12243.215} C_VEL
LIN {X 0,Y 376.237,Z 270.427,A -85,B 0,C 180,E1 -12246.437,E2 -12246.437} C_VEL
LIN {X 0,Y 376.196,Z 270.44,A -85,B 0,C 180,E1 -12248.597,E2 -12248.597} C_VEL
LIN {X 0,Y 376.048,Z 270.459,A -85,B 0,C 180,E1 -12251.865,E2 -12251.865} C_VEL
LIN {X 0,Y 376.051,Z 270.457,A -85,B 0,C 180,E1 -12255.169,E2 -12255.169} C_VEL
LIN {X 0,Y 376.015,Z 270.46,A -85,B 0,C 180,E1 -12258.528,E2 -12258.528} C_VEL
LIN {X 0,Y 375.949,Z 270.467,A -85,B 0,C 180,E1 -12261.957,E2 -12261.957} C_VEL
LIN {X 0,Y 375.959,Z 270.468,A -85,B 0,C 180,E1 -12265.466,E2 -12265.466} C_VEL
LIN {X 0,Y 375.913,Z 270.478,A -85,B 0,C 180,E1 -12269.085,E2 -12269.085} C_VEL
LIN {X 0,Y 375.952,Z 270.471,A -85,B 0,C 180,E1 -12271.564,E2 -12271.564} C_VEL
LIN {X 0,Y 375.952,Z 270.473,A -85,B 0,C 180,E1 -12275.418,E2 -12275.418} C_VEL
LIN {X 0,Y 375.972,Z 270.467,A -85,B 0,C 180,E1 -12278.273,E2 -12278.273} C_VEL
LIN {X 0,Y 375.956,Z 270.469,A -85,B 0,C 180,E1 -12281.607,E2 -12281.607} C_VEL
LIN {X 0,Y 375.924,Z 270.475,A -85,B 0,C 180,E1 -12285.271,E2 -12285.271} C_VEL
LIN {X 0,Y 376.01,Z 270.59,A -85,B 0,C 180,E1 -12288.996,E2 -12288.996} C_VEL
LIN {X 0,Y 376.799,Z 275.179,A -85,B 0,C 180,E1 -12292.013,E2 -12292.013} C_VEL
LIN {X 0,Y 377.593,Z 279.993,A -85,B 0,C 180,E1 -12294.982,E2 -12294.982} C_VEL
LIN {X 0,Y 377.915,Z 283.125,A -85,B 0,C 180,E1 -12296.811,E2 -12296.811} C_VEL
LIN {X 0,Y 377.321,Z 288.649,A -85,B 0,C 180,E1 -12299.81,E2 -12299.81} C_VEL
LIN {X 0,Y 376.455,Z 296.074,A -85,B 0,C 180,E1 -12303.653,E2 -12303.653} C_VEL
LIN {X 0,Y 375.863,Z 302.542,A -85,B 0,C 180,E1 -12306.881,E2 -12306.881} C_VEL
LIN {X 0,Y 375.308,Z 310.73,A -85,B 0,C 180,E1 -12310.872,E2 -12310.872} C_VEL
LIN {X 0,Y 374.98,Z 317.578,A -85,B 0,C 180,E1 -12314.128,E2 -12314.128} C_VEL
LIN {X 0,Y 377.032,Z 329.795,A -85,B 0,C 180,E1 -12314.736,E2 -12314.736} C_VEL
LIN {X 0,Y 378.145,Z 340.173,A -85,B 0,C 180,E1 -12315.438,E2 -12315.438} C_VEL
LIN {X 0,Y 378.449,Z 347.503,A -85,B 0,C 180,E1 -12316.031,E2 -12316.031} C_VEL
LIN {X 0,Y 377.934,Z 355.903,A -85,B 0,C 180,E1 -12316.834,E2 -12316.834} C_VEL
LIN {X 0,Y 377.183,Z 363.858,A -85,B 0,C 180,E1 -12317.765,E2 -12317.765} C_VEL
LIN {X 0,Y 376.527,Z 370.448,A -85,B 0,C 180,E1 -12318.699,E2 -12318.699} C_VEL
LIN {X 0,Y 375.927,Z 376.725,A -85,B 0,C 180,E1 -12319.771,E2 -12319.771} C_VEL
LIN {X 0,Y 375.447,Z 381.954,A -85,B 0,C 180,E1 -12320.846,E2 -12320.846} C_VEL
LIN {X 0,Y 375.098,Z 386.33,A -85,B 0,C 180,E1 -12321.923,E2 -12321.923} C_VEL
LIN {X 0,Y 374.73,Z 391.513,A -85,B 0,C 180,E1 -12323.54,E2 -12323.54} C_VEL
LIN {X 0,Y 374.616,Z 395.336,A -85,B 0,C 180,E1 -12325.159,E2 -12325.159} C_VEL
LIN {X 0,Y 374.51,Z 397.87,A -85,B 0,C 180,E1 -12326.774,E2 -12326.774} C_VEL
LIN {X 0,Y 374.556,Z 398.869,A -85,B 0,C 180,E1 -12327.851,E2 -12327.851} C_VEL
LIN {X 0,Y 374.624,Z 399.35,A -85,B 0,C 180,E1 -12328.926,E2 -12328.926} C_VEL
LIN {X 0,Y 374.61,Z 399.366,A -85,B 0,C 180,E1 -12330.001,E2 -12330.001} C_VEL
LIN {X 0,Y 374.627,Z 398.92,A -85,B 0,C 180,E1 -12331.076,E2 -12331.076} C_VEL
LIN {X 0,Y 374.599,Z 397.948,A -85,B 0,C 180,E1 -12332.152,E2 -12332.152} C_VEL
LIN {X 0,Y 374.556,Z 395.428,A -85,B 0,C 180,E1 -12333.767,E2 -12333.767} C_VEL
LIN {X 0,Y 374.635,Z 393.093,A -85,B 0,C 180,E1 -12334.844,E2 -12334.844} C_VEL
LIN {X 0,Y 374.732,Z 388.307,A -85,B 0,C 180,E1 -12336.462,E2 -12336.462} C_VEL
LIN {X 0,Y 374.969,Z 383.118,A -85,B 0,C 180,E1 -12337.811,E2 -12337.811} C_VEL
LIN {X 0,Y 375.235,Z 378.038,A -85,B 0,C 180,E1 -12338.89,E2 -12338.89} C_VEL
LIN {X 0,Y 375.593,Z 371.913,A -85,B 0,C 180,E1 -12339.968,E2 -12339.968} C_VEL
LIN {X 0,Y 376.052,Z 364.456,A -85,B 0,C 180,E1 -12341.045,E2 -12341.045} C_VEL
LIN {X 0,Y 376.545,Z 356.46,A -85,B 0,C 180,E1 -12341.985,E2 -12341.985} C_VEL
LIN {X 0,Y 377.083,Z 348,A -85,B 0,C 180,E1 -12342.788,E2 -12342.788} C_VEL
LIN {X 0,Y 376.527,Z 336.854,A -85,B 0,C 180,E1 -12343.631,E2 -12343.631} C_VEL
LIN {X 0,Y 375.535,Z 326.032,A -85,B 0,C 180,E1 -12344.22,E2 -12344.22} C_VEL
LIN {X 0,Y 374.764,Z 317.962,A -85,B 0,C 180,E1 -12344.562,E2 -12344.562} C_VEL
LIN {X 0,Y 375.021,Z 310.494,A -85,B 0,C 180,E1 -12348.013,E2 -12348.013} C_VEL
LIN {X 0,Y 375.496,Z 301.994,A -85,B 0,C 180,E1 -12351.984,E2 -12351.984} C_VEL
LIN {X 0,Y 376.113,Z 293.045,A -85,B 0,C 180,E1 -12356.242,E2 -12356.242} C_VEL
LIN {X 0,Y 376.819,Z 284.902,A -85,B 0,C 180,E1 -12360.238,E2 -12360.238} C_VEL
LIN {X 0,Y 377.327,Z 279.318,A -85,B 0,C 180,E1 -12363.052,E2 -12363.052} C_VEL
LIN {X 0,Y 376.835,Z 275.067,A -85,B 0,C 180,E1 -12365.322,E2 -12365.322} C_VEL
LIN {X 0,Y 376.015,Z 270.462,A -85,B 0,C 180,E1 -12367.914,E2 -12367.914} C_VEL
LIN {X 0,Y 375.949,Z 270.466,A -85,B 0,C 180,E1 -12370.867,E2 -12370.867} C_VEL
LIN {X 0,Y 375.939,Z 270.471,A -85,B 0,C 180,E1 -12373.766,E2 -12373.766} C_VEL
LIN {X 0,Y 375.943,Z 270.466,A -85,B 0,C 180,E1 -12376.811,E2 -12376.811} C_VEL
LIN {X 0,Y 375.97,Z 270.464,A -85,B 0,C 180,E1 -12380.537,E2 -12380.537} C_VEL
LIN {X 0,Y 375.973,Z 270.467,A -85,B 0,C 180,E1 -12383.495,E2 -12383.495} C_VEL
LIN {X 0,Y 375.97,Z 270.467,A -85,B 0,C 180,E1 -12385.888,E2 -12385.888} C_VEL
LIN {X 0,Y 375.974,Z 270.467,A -85,B 0,C 180,E1 -12389.687,E2 -12389.687} C_VEL
LIN {X 0,Y 376.006,Z 270.459,A -85,B 0,C 180,E1 -12392.141,E2 -12392.141} C_VEL
LIN {X 0,Y 376.015,Z 270.458,A -85,B 0,C 180,E1 -12394.538,E2 -12394.538} C_VEL
LIN {X 0,Y 375.967,Z 270.464,A -85,B 0,C 180,E1 -12398.044,E2 -12398.044} C_VEL
LIN {X 0,Y 376.012,Z 270.461,A -85,B 0,C 180,E1 -12401.472,E2 -12401.472} C_VEL
LIN {X 0,Y 376.067,Z 270.455,A -85,B 0,C 180,E1 -12404.831,E2 -12404.831} C_VEL
LIN {X 0,Y 376.057,Z 270.453,A -85,B 0,C 180,E1 -12408.135,E2 -12408.135} C_VEL
LIN {X 0,Y 376.207,Z 270.434,A -85,B 0,C 180,E1 -12411.938,E2 -12411.938} C_VEL
LIN {X 0,Y 376.173,Z 270.442,A -85,B 0,C 180,E1 -12414.638,E2 -12414.638} C_VEL
LIN {X 0,Y 376.358,Z 270.415,A -85,B 0,C 180,E1 -12417.858,E2 -12417.858} C_VEL
LIN {X 0,Y 376.493,Z 270.399,A -85,B 0,C 180,E1 -12419.998,E2 -12419.998} C_VEL
LIN {X 0,Y 376.194,Z 270.436,A -85,B 0,C 180,E1 -12423.211,E2 -12423.211} C_VEL
LIN {X 0,Y 376.24,Z 270.432,A -85,B 0,C 180,E1 -12426.601,E2 -12426.601} C_VEL
LIN {X 0,Y 376.21,Z 270.437,A -85,B 0,C 180,E1 -12428.593,E2 -12428.593} C_VEL
LIN {X 0,Y 376.053,Z 270.455,A -85,B 0,C 180,E1 -12431.861,E2 -12431.861} C_VEL
LIN {X 0,Y 376.061,Z 270.452,A -85,B 0,C 180,E1 -12435.165,E2 -12435.165} C_VEL
LIN {X 0,Y 376.025,Z 270.458,A -85,B 0,C 180,E1 -12438.524,E2 -12438.524} C_VEL
LIN {X 0,Y 375.963,Z 270.469,A -85,B 0,C 180,E1 -12441.952,E2 -12441.952} C_VEL
LIN {X 0,Y 376.005,Z 270.461,A -85,B 0,C 180,E1 -12445.458,E2 -12445.458} C_VEL
LIN {X 0,Y 375.959,Z 270.465,A -85,B 0,C 180,E1 -12449.077,E2 -12449.077} C_VEL
LIN {X 0,Y 375.945,Z 270.466,A -85,B 0,C 180,E1 -12452.826,E2 -12452.826} C_VEL
LIN {X 0,Y 375.954,Z 270.469,A -85,B 0,C 180,E1 -12455.413,E2 -12455.413} C_VEL
LIN {X 0,Y 375.972,Z 270.463,A -85,B 0,C 180,E1 -12458.268,E2 -12458.268} C_VEL
LIN {X 0,Y 375.983,Z 270.465,A -85,B 0,C 180,E1 -12461.608,E2 -12461.608} C_VEL
LIN {X 0,Y 376.007,Z 270.463,A -85,B 0,C 180,E1 -12465.252,E2 -12465.252} C_VEL
LIN {X 0,Y 375.991,Z 270.465,A -85,B 0,C 180,E1 -12469.138,E2 -12469.138} C_VEL
LIN {X 0,Y 375.958,Z 270.465,A -85,B 0,C 180,E1 -12471.909,E2 -12471.909} C_VEL
LIN {X 0,Y 375.969,Z 270.466,A -85,B 0,C 180,E1 -12475.33,E2 -12475.33} C_VEL
LIN {X 0,Y 375.947,Z 270.468,A -85,B 0,C 180,E1 -12478.436,E2 -12478.436} C_VEL
LIN {X 0,Y 375.989,Z 270.462,A -85,B 0,C 180,E1 -12482.139,E2 -12482.139} C_VEL
LIN {X 0,Y 375.993,Z 270.464,A -85,B 0,C 180,E1 -12484.537,E2 -12484.537} C_VEL
LIN {X 0,Y 375.965,Z 270.465,A -85,B 0,C 180,E1 -12488.045,E2 -12488.045} C_VEL
LIN {X 0,Y 375.884,Z 270.474,A -85,B 0,C 180,E1 -12491.466,E2 -12491.466} C_VEL
LIN {X 0,Y 375.636,Z 270.506,A -85,B 0,C 180,E1 -12493.7,E2 -12493.7} C_VEL
LIN {X 0,Y 375.363,Z 270.544,A -85,B 0,C 180,E1 -12495.911,E2 -12495.911} C_VEL
LIN {X 0,Y 375.316,Z 272.882,A -85,B 0,C 180,E1 -12498.112,E2 -12498.112} C_VEL
LIN {X 0,Y 375.208,Z 276.589,A -85,B 0,C 180,E1 -12501.381,E2 -12501.381} C_VEL
LIN {X 0,Y 375.26,Z 279.068,A -85,B 0,C 180,E1 -12503.547,E2 -12503.547} C_VEL
LIN {X 0,Y 375.101,Z 282.853,A -85,B 0,C 180,E1 -12506.776,E2 -12506.776} C_VEL
LIN {X 0,Y 374.888,Z 286.207,A -85,B 0,C 180,E1 -12509.596,E2 -12509.596} C_VEL
LIN {X 0,Y 376.637,Z 297.064,A -85,B 0,C 180,E1 -12510.132,E2 -12510.132} C_VEL
LIN {X 0,Y 377.923,Z 305.233,A -85,B 0,C 180,E1 -12510.665,E2 -12510.665} C_VEL
LIN {X 0,Y 377.582,Z 313.937,A -85,B 0,C 180,E1 -12511.332,E2 -12511.332} C_VEL
LIN {X 0,Y 377.126,Z 322.277,A -85,B 0,C 180,E1 -12512.135,E2 -12512.135} C_VEL
LIN {X 0,Y 376.603,Z 330.182,A -85,B 0,C 180,E1 -12513.074,E2 -12513.074} C_VEL
LIN {X 0,Y 376.193,Z 336.695,A -85,B 0,C 180,E1 -12514.016,E2 -12514.016} C_VEL
LIN {X 0,Y 375.783,Z 342.893,A -85,B 0,C 180,E1 -12515.095,E2 -12515.095} C_VEL
LIN {X 0,Y 375.554,Z 348.02,A -85,B 0,C 180,E1 -12516.176,E2 -12516.176} C_VEL
LIN {X 0,Y 375.192,Z 353.28,A -85,B 0,C 180,E1 -12517.533,E2 -12517.533} C_VEL
LIN {X 0,Y 374.844,Z 358.163,A -85,B 0,C 180,E1 -12519.169,E2 -12519.169} C_VEL
LIN {X 0,Y 374.648,Z 361.521,A -85,B 0,C 180,E1 -12520.811,E2 -12520.811} C_VEL
LIN {X 0,Y 374.564,Z 363.133,A -85,B 0,C 180,E1 -12521.91,E2 -12521.91} C_VEL
LIN {X 0,Y 374.512,Z 364.14,A -85,B 0,C 180,E1 -12523.012,E2 -12523.012} C_VEL
LIN {X 0,Y 374.468,Z 364.61,A -85,B 0,C 180,E1 -12524.12,E2 -12524.12} C_VEL
LIN {X 0,Y 374.507,Z 364.586,A -85,B 0,C 180,E1 -12525.23,E2 -12525.23} C_VEL
LIN {X 0,Y 374.708,Z 363.524,A -85,B 0,C 180,E1 -12526.962,E2 -12526.962} C_VEL
LIN {X 0,Y 374.968,Z 361.383,A -85,B 0,C 180,E1 -12528.578,E2 -12528.578} C_VEL
LIN {X 0,Y 375.376,Z 358.028,A -85,B 0,C 180,E1 -12530.17,E2 -12530.17} C_VEL
LIN {X 0,Y 375.697,Z 354.575,A -85,B 0,C 180,E1 -12531.392,E2 -12531.392} C_VEL
LIN {X 0,Y 376.219,Z 349.416,A -85,B 0,C 180,E1 -12532.805,E2 -12532.805} C_VEL
LIN {X 0,Y 376.915,Z 342.846,A -85,B 0,C 180,E1 -12534.217,E2 -12534.217} C_VEL
LIN {X 0,Y 377.332,Z 338.092,A -85,B 0,C 180,E1 -12535.069,E2 -12535.069} C_VEL
LIN {X 0,Y 378.098,Z 330.446,A -85,B 0,C 180,E1 -12536.195,E2 -12536.195} C_VEL
LIN {X 0,Y 378.743,Z 323.407,A -85,B 0,C 180,E1 -12537.046,E2 -12537.046} C_VEL
LIN {X 0,Y 379.397,Z 314.978,A -85,B 0,C 180,E1 -12537.878,E2 -12537.878} C_VEL
LIN {X 0,Y 379.664,Z 308.03,A -85,B 0,C 180,E1 -12538.444,E2 -12538.444} C_VEL
LIN {X 0,Y 378.063,Z 299.248,A -85,B 0,C 180,E1 -12539.114,E2 -12539.114} C_VEL
LIN {X 0,Y 377.449,Z 296.583,A -85,B 0,C 180,E1 -12539.303,E2 -12539.303} C_VEL
LIN {X 0,Y 375.951,Z 293.261,A -85,B 0,C 180,E1 -12539.601,E2 -12539.601} C_VEL
LIN {X 0,Y 373.715,Z 290.601,A -85,B 0,C 180,E1 -12539.959,E2 -12539.959} C_VEL
LIN {X 0,Y 370.571,Z 287.92,A -85,B 0,C 180,E1 -12540.534,E2 -12540.534} C_VEL
LIN {X 0,Y 368.48,Z 286.257,A -85,B 0,C 180,E1 -12541.15,E2 -12541.15} C_VEL
LIN {X 0,Y 367.919,Z 285.476,A -85,B 0,C 180,E1 -12541.652,E2 -12541.652} C_VEL
LIN {X 0,Y 368.019,Z 281.913,A -85,B 0,C 180,E1 -12544.951,E2 -12544.951} C_VEL
LIN {X 0,Y 368.204,Z 279.065,A -85,B 0,C 180,E1 -12547.645,E2 -12547.645} C_VEL
LIN {X 0,Y 368.39,Z 276.168,A -85,B 0,C 180,E1 -12550.437,E2 -12550.437} C_VEL
LIN {X 0,Y 368.552,Z 272.995,A -85,B 0,C 180,E1 -12553.566,E2 -12553.566} C_VEL
LIN {X 0,Y 368.605,Z 271.456,A -85,B 0,C 180,E1 -12555.137,E2 -12555.137} C_VEL
LIN {X 0,Y 368.808,Z 271.359,A -85,B 0,C 180,E1 -12558.171,E2 -12558.171} C_VEL
LIN {X 0,Y 368.891,Z 271.351,A -85,B 0,C 180,E1 -12561.36,E2 -12561.36} C_VEL
LIN {X 0,Y 368.918,Z 271.345,A -85,B 0,C 180,E1 -12565.148,E2 -12565.148} C_VEL
LIN {X 0,Y 368.911,Z 271.346,A -85,B 0,C 180,E1 -12569.048,E2 -12569.048} C_VEL
LIN {X 0,Y 368.945,Z 271.34,A -85,B 0,C 180,E1 -12572.798,E2 -12572.798} C_VEL
LIN {X 0,Y 368.92,Z 271.34,A -85,B 0,C 180,E1 -12576.117,E2 -12576.117} C_VEL
LIN {X 0,Y 368.921,Z 271.343,A -85,B 0,C 180,E1 -12579.949,E2 -12579.949} C_VEL
LIN {X 0,Y 368.961,Z 271.34,A -85,B 0,C 180,E1 -12583.4,E2 -12583.4} C_VEL
LIN {X 0,Y 369.045,Z 271.328,A -85,B 0,C 180,E1 -12586.792,E2 -12586.792} C_VEL
LIN {X 0,Y 369.058,Z 271.324,A -85,B 0,C 180,E1 -12590.134,E2 -12590.134} C_VEL
LIN {X 0,Y 369.16,Z 271.308,A -85,B 0,C 180,E1 -12593.443,E2 -12593.443} C_VEL
LIN {X 0,Y 369.308,Z 271.291,A -85,B 0,C 180,E1 -12597.821,E2 -12597.821} C_VEL
LIN {X 0,Y 369.446,Z 271.277,A -85,B 0,C 180,E1 -12600.002,E2 -12600.002} C_VEL
LIN {X 0,Y 369.305,Z 271.292,A -85,B 0,C 180,E1 -12602.183,E2 -12602.183} C_VEL
LIN {X 0,Y 369.199,Z 271.304,A -85,B 0,C 180,E1 -12606.56,E2 -12606.56} C_VEL
LIN {X 0,Y 369.128,Z 271.319,A -85,B 0,C 180,E1 -12608.763,E2 -12608.763} C_VEL
LIN {X 0,Y 369.003,Z 271.334,A -85,B 0,C 180,E1 -12612.095,E2 -12612.095} C_VEL
LIN {X 0,Y 368.99,Z 271.335,A -85,B 0,C 180,E1 -12615.467,E2 -12615.467} C_VEL
LIN {X 0,Y 368.958,Z 271.338,A -85,B 0,C 180,E1 -12618.896,E2 -12618.896} C_VEL
LIN {X 0,Y 368.914,Z 271.344,A -85,B 0,C 180,E1 -12622.398,E2 -12622.398} C_VEL
LIN {X 0,Y 368.937,Z 271.346,A -85,B 0,C 180,E1 -12625.987,E2 -12625.987} C_VEL
LIN {X 0,Y 368.89,Z 271.351,A -85,B 0,C 180,E1 -12629.694,E2 -12629.694} C_VEL
LIN {X 0,Y 368.892,Z 271.351,A -85,B 0,C 180,E1 -12633.045,E2 -12633.045} C_VEL
LIN {X 0,Y 368.912,Z 271.347,A -85,B 0,C 180,E1 -12636.199,E2 -12636.199} C_VEL
LIN {X 0,Y 368.903,Z 271.348,A -85,B 0,C 180,E1 -12638.955,E2 -12638.955} C_VEL
LIN {X 0,Y 368.906,Z 271.348,A -85,B 0,C 180,E1 -12642.016,E2 -12642.016} C_VEL
LIN {X 0,Y 368.877,Z 271.354,A -85,B 0,C 180,E1 -12645.178,E2 -12645.178} C_VEL
LIN {X 0,Y 368.919,Z 271.424,A -85,B 0,C 180,E1 -12648.55,E2 -12648.55} C_VEL
LIN {X 0,Y 369.824,Z 276.362,A -85,B 0,C 180,E1 -12651.901,E2 -12651.901} C_VEL
LIN {X 0,Y 370.68,Z 281.841,A -85,B 0,C 180,E1 -12655.336,E2 -12655.336} C_VEL
LIN {X 0,Y 370.815,Z 285.222,A -85,B 0,C 180,E1 -12657.308,E2 -12657.308} C_VEL
LIN {X 0,Y 370.028,Z 291.779,A -85,B 0,C 180,E1 -12660.892,E2 -12660.892} C_VEL
LIN {X 0,Y 369.219,Z 298.939,A -85,B 0,C 180,E1 -12664.643,E2 -12664.643} C_VEL
LIN {X 0,Y 368.568,Z 305.918,A -85,B 0,C 180,E1 -12668.173,E2 -12668.173} C_VEL
LIN {X 0,Y 368.126,Z 314.088,A -85,B 0,C 180,E1 -12672.216,E2 -12672.216} C_VEL
LIN {X 0,Y 367.935,Z 317.277,A -85,B 0,C 180,E1 -12673.744,E2 -12673.744} C_VEL
LIN {X 0,Y 370.016,Z 329.434,A -85,B 0,C 180,E1 -12674.369,E2 -12674.369} C_VEL
LIN {X 0,Y 371.195,Z 339.802,A -85,B 0,C 180,E1 -12675.089,E2 -12675.089} C_VEL
LIN {X 0,Y 371.564,Z 347.878,A -85,B 0,C 180,E1 -12675.767,E2 -12675.767} C_VEL
LIN {X 0,Y 371.047,Z 356.149,A -85,B 0,C 180,E1 -12676.585,E2 -12676.585} C_VEL
LIN {X 0,Y 370.338,Z 362.988,A -85,B 0,C 180,E1 -12677.396,E2 -12677.396} C_VEL
LIN {X 0,Y 369.729,Z 368.813,A -85,B 0,C 180,E1 -12678.211,E2 -12678.211} C_VEL
LIN {X 0,Y 369.101,Z 375.306,A -85,B 0,C 180,E1 -12679.303,E2 -12679.303} C_VEL
LIN {X 0,Y 368.559,Z 380.722,A -85,B 0,C 180,E1 -12680.397,E2 -12680.397} C_VEL
LIN {X 0,Y 368.05,Z 386.22,A -85,B 0,C 180,E1 -12681.768,E2 -12681.768} C_VEL
LIN {X 0,Y 367.654,Z 391.354,A -85,B 0,C 180,E1 -12683.415,E2 -12683.415} C_VEL
LIN {X 0,Y 367.531,Z 395.132,A -85,B 0,C 180,E1 -12685.065,E2 -12685.065} C_VEL
LIN {X 0,Y 367.427,Z 397.598,A -85,B 0,C 180,E1 -12686.712,E2 -12686.712} C_VEL
LIN {X 0,Y 367.455,Z 398.59,A -85,B 0,C 180,E1 -12687.809,E2 -12687.809} C_VEL
LIN {X 0,Y 367.538,Z 399.036,A -85,B 0,C 180,E1 -12688.906,E2 -12688.906} C_VEL
LIN {X 0,Y 367.544,Z 399.019,A -85,B 0,C 180,E1 -12690.001,E2 -12690.001} C_VEL
LIN {X 0,Y 367.561,Z 398.539,A -85,B 0,C 180,E1 -12691.097,E2 -12691.097} C_VEL
LIN {X 0,Y 367.501,Z 397.552,A -85,B 0,C 180,E1 -12692.193,E2 -12692.193} C_VEL
LIN {X 0,Y 367.482,Z 394.974,A -85,B 0,C 180,E1 -12693.839,E2 -12693.839} C_VEL
LIN {X 0,Y 367.547,Z 392.618,A -85,B 0,C 180,E1 -12694.938,E2 -12694.938} C_VEL
LIN {X 0,Y 367.658,Z 387.767,A -85,B 0,C 180,E1 -12696.587,E2 -12696.587} C_VEL
LIN {X 0,Y 367.887,Z 383.716,A -85,B 0,C 180,E1 -12697.686,E2 -12697.686} C_VEL
LIN {X 0,Y 368.181,Z 377.39,A -85,B 0,C 180,E1 -12699.062,E2 -12699.062} C_VEL
LIN {X 0,Y 368.556,Z 371.198,A -85,B 0,C 180,E1 -12700.161,E2 -12700.161} C_VEL
LIN {X 0,Y 368.992,Z 364.693,A -85,B 0,C 180,E1 -12701.12,E2 -12701.12} C_VEL
LIN {X 0,Y 369.491,Z 356.807,A -85,B 0,C 180,E1 -12702.078,E2 -12702.078} C_VEL
LIN {X 0,Y 369.995,Z 350.007,A -85,B 0,C 180,E1 -12702.758,E2 -12702.758} C_VEL
LIN {X 0,Y 369.826,Z 342.352,A -85,B 0,C 180,E1 -12703.405,E2 -12703.405} C_VEL
LIN {X 0,Y 369.167,Z 333.597,A -85,B 0,C 180,E1 -12704.006,E2 -12704.006} C_VEL
LIN {X 0,Y 368.33,Z 324.036,A -85,B 0,C 180,E1 -12704.505,E2 -12704.505} C_VEL
LIN {X 0,Y 367.677,Z 317.662,A -85,B 0,C 180,E1 -12704.778,E2 -12704.778} C_VEL
LIN {X 0,Y 367.982,Z 310.059,A -85,B 0,C 180,E1 -12708.37,E2 -12708.37} C_VEL
LIN {X 0,Y 368.462,Z 301.579,A -85,B 0,C 180,E1 -12712.427,E2 -12712.427} C_VEL
LIN {X 0,Y 369.074,Z 293.238,A -85,B 0,C 180,E1 -12716.491,E2 -12716.491} C_VEL
LIN {X 0,Y 369.772,Z 285.76,A -85,B 0,C 180,E1 -12720.244,E2 -12720.244} C_VEL
LIN {X 0,Y 370.274,Z 280.9,A -85,B 0,C 180,E1 -12722.732,E2 -12722.732} C_VEL
LIN {X 0,Y 369.98,Z 277.183,A -85,B 0,C 180,E1 -12724.742,E2 -12724.742} C_VEL
LIN {X 0,Y 368.989,Z 271.337,A -85,B 0,C 180,E1 -12728.072,E2 -12728.072} C_VEL
LIN {X 0,Y 368.892,Z 271.349,A -85,B 0,C 180,E1 -12731.823,E2 -12731.823} C_VEL
LIN {X 0,Y 368.889,Z 271.345,A -85,B 0,C 180,E1 -12735.176,E2 -12735.176} C_VEL
LIN {X 0,Y 368.892,Z 271.348,A -85,B 0,C 180,E1 -12738.177,E2 -12738.177} C_VEL
LIN {X 0,Y 368.915,Z 271.344,A -85,B 0,C 180,E1 -12741.36,E2 -12741.36} C_VEL
LIN {X 0,Y 368.946,Z 271.34,A -85,B 0,C 180,E1 -12745.146,E2 -12745.146} C_VEL
LIN {X 0,Y 368.939,Z 271.341,A -85,B 0,C 180,E1 -12749.046,E2 -12749.046} C_VEL
LIN {X 0,Y 368.99,Z 271.337,A -85,B 0,C 180,E1 -12751.563,E2 -12751.563} C_VEL
LIN {X 0,Y 369.009,Z 271.331,A -85,B 0,C 180,E1 -12754.019,E2 -12754.019} C_VEL
LIN {X 0,Y 368.934,Z 271.342,A -85,B 0,C 180,E1 -12757.603,E2 -12757.603} C_VEL
LIN {X 0,Y 368.963,Z 271.341,A -85,B 0,C 180,E1 -12761.105,E2 -12761.105} C_VEL
LIN {X 0,Y 369.006,Z 271.332,A -85,B 0,C 180,E1 -12764.534,E2 -12764.534} C_VEL
LIN {X 0,Y 369.012,Z 271.33,A -85,B 0,C 180,E1 -12767.905,E2 -12767.905} C_VEL
LIN {X 0,Y 369.154,Z 271.312,A -85,B 0,C 180,E1 -12771.889,E2 -12771.889} C_VEL
LIN {X 0,Y 369.145,Z 271.317,A -85,B 0,C 180,E1 -12774.536,E2 -12774.536} C_VEL
LIN {X 0,Y 369.323,Z 271.291,A -85,B 0,C 180,E1 -12777.817,E2 -12777.817} C_VEL
LIN {X 0,Y 369.463,Z 271.275,A -85,B 0,C 180,E1 -12779.998,E2 -12779.998} C_VEL
LIN {X 0,Y 369.325,Z 271.293,A -85,B 0,C 180,E1 -12782.179,E2 -12782.179} C_VEL
LIN {X 0,Y 369.211,Z 271.309,A -85,B 0,C 180,E1 -12786.589,E2 -12786.589} C_VEL
LIN {X 0,Y 369.142,Z 271.316,A -85,B 0,C 180,E1 -12788.759,E2 -12788.759} C_VEL
LIN {X 0,Y 369.009,Z 271.334,A -85,B 0,C 180,E1 -12792.091,E2 -12792.091} C_VEL
LIN {X 0,Y 369,Z 271.332,A -85,B 0,C 180,E1 -12795.462,E2 -12795.462} C_VEL
LIN {X 0,Y 368.968,Z 271.336,A -85,B 0,C 180,E1 -12798.891,E2 -12798.891} C_VEL
LIN {X 0,Y 368.932,Z 271.342,A -85,B 0,C 180,E1 -12802.392,E2 -12802.392} C_VEL
LIN {X 0,Y 368.999,Z 271.336,A -85,B 0,C 180,E1 -12805.977,E2 -12805.977} C_VEL
LIN {X 0,Y 368.912,Z 271.347,A -85,B 0,C 180,E1 -12809.688,E2 -12809.688} C_VEL
LIN {X 0,Y 368.893,Z 271.346,A -85,B 0,C 180,E1 -12813.04,E2 -12813.04} C_VEL
LIN {X 0,Y 368.914,Z 271.343,A -85,B 0,C 180,E1 -12816.194,E2 -12816.194} C_VEL
LIN {X 0,Y 368.903,Z 271.345,A -85,B 0,C 180,E1 -12818.95,E2 -12818.95} C_VEL
LIN {X 0,Y 368.935,Z 271.34,A -85,B 0,C 180,E1 -12822.017,E2 -12822.017} C_VEL
LIN {X 0,Y 368.982,Z 271.338,A -85,B 0,C 180,E1 -12825.19,E2 -12825.19} C_VEL
LIN {X 0,Y 368.932,Z 271.34,A -85,B 0,C 180,E1 -12828.183,E2 -12828.183} C_VEL
LIN {X 0,Y 368.904,Z 271.346,A -85,B 0,C 180,E1 -12831.356,E2 -12831.356} C_VEL
LIN {X 0,Y 368.925,Z 271.345,A -85,B 0,C 180,E1 -12835.144,E2 -12835.144} C_VEL
LIN {X 0,Y 368.917,Z 271.346,A -85,B 0,C 180,E1 -12839.044,E2 -12839.044} C_VEL
LIN {X 0,Y 368.974,Z 271.335,A -85,B 0,C 180,E1 -12841.562,E2 -12841.562} C_VEL
LIN {X 0,Y 368.946,Z 271.339,A -85,B 0,C 180,E1 -12845.222,E2 -12845.222} C_VEL
LIN {X 0,Y 368.956,Z 271.339,A -85,B 0,C 180,E1 -12848.958,E2 -12848.958} C_VEL
LIN {X 0,Y 368.784,Z 271.363,A -85,B 0,C 180,E1 -12852.327,E2 -12852.327} C_VEL
LIN {X 0,Y 368.359,Z 271.414,A -85,B 0,C 180,E1 -12855.638,E2 -12855.638} C_VEL
LIN {X 0,Y 368.352,Z 272.103,A -85,B 0,C 180,E1 -12856.763,E2 -12856.763} C_VEL
LIN {X 0,Y 368.16,Z 277.076,A -85,B 0,C 180,E1 -12861.214,E2 -12861.214} C_VEL
LIN {X 0,Y 368.22,Z 279.574,A -85,B 0,C 180,E1 -12863.423,E2 -12863.423} C_VEL
LIN {X 0,Y 368.041,Z 283.382,A -85,B 0,C 180,E1 -12866.714,E2 -12866.714} C_VEL
LIN {X 0,Y 367.824,Z 286.534,A -85,B 0,C 180,E1 -12869.383,E2 -12869.383} C_VEL
LIN {X 0,Y 369.604,Z 297.423,A -85,B 0,C 180,E1 -12869.93,E2 -12869.93} C_VEL
LIN {X 0,Y 370.944,Z 306.472,A -85,B 0,C 180,E1 -12870.541,E2 -12870.541} C_VEL
LIN {X 0,Y 370.541,Z 315.013,A -85,B 0,C 180,E1 -12871.221,E2 -12871.221} C_VEL
LIN {X 0,Y 370.082,Z 323.216,A -85,B 0,C 180,E1 -12872.039,E2 -12872.039} C_VEL
LIN {X 0,Y 369.544,Z 331.018,A -85,B 0,C 180,E1 -12872.996,E2 -12872.996} C_VEL
LIN {X 0,Y 369.09,Z 338.298,A -85,B 0,C 180,E1 -12874.093,E2 -12874.093} C_VEL
LIN {X 0,Y 368.553,Z 345.683,A -85,B 0,C 180,E1 -12875.47,E2 -12875.47} C_VEL
LIN {X 0,Y 368.38,Z 350.405,A -85,B 0,C 180,E1 -12876.571,E2 -12876.571} C_VEL
LIN {X 0,Y 367.939,Z 356.01,A -85,B 0,C 180,E1 -12878.235,E2 -12878.235} C_VEL
LIN {X 0,Y 367.64,Z 360.14,A -85,B 0,C 180,E1 -12879.905,E2 -12879.905} C_VEL
LIN {X 0,Y 367.534,Z 362.163,A -85,B 0,C 180,E1 -12881.022,E2 -12881.022} C_VEL
LIN {X 0,Y 367.448,Z 364.186,A -85,B 0,C 180,E1 -12882.736,E2 -12882.736} C_VEL
LIN {X 0,Y 367.403,Z 365.006,A -85,B 0,C 180,E1 -12884.398,E2 -12884.398} C_VEL
LIN {X 0,Y 367.451,Z 364.859,A -85,B 0,C 180,E1 -12885.53,E2 -12885.53} C_VEL
LIN {X 0,Y 367.636,Z 363.84,A -85,B 0,C 180,E1 -12887.102,E2 -12887.102} C_VEL
LIN {X 0,Y 367.971,Z 361.352,A -85,B 0,C 180,E1 -12888.945,E2 -12888.945} C_VEL
LIN {X 0,Y 368.371,Z 358.037,A -85,B 0,C 180,E1 -12890.472,E2 -12890.472} C_VEL
LIN {X 0,Y 368.766,Z 354.17,A -85,B 0,C 180,E1 -12891.815,E2 -12891.815} C_VEL
LIN {X 0,Y 369.376,Z 348.835,A -85,B 0,C 180,E1 -12893.252,E2 -12893.252} C_VEL
LIN {X 0,Y 369.934,Z 343.796,A -85,B 0,C 180,E1 -12894.354,E2 -12894.354} C_VEL
LIN {X 0,Y 370.418,Z 338.869,A -85,B 0,C 180,E1 -12895.269,E2 -12895.269} C_VEL
LIN {X 0,Y 371.206,Z 331.31,A -85,B 0,C 180,E1 -12896.417,E2 -12896.417} C_VEL
LIN {X 0,Y 371.83,Z 324.892,A -85,B 0,C 180,E1 -12897.226,E2 -12897.226} C_VEL
LIN {X 0,Y 372.492,Z 317.401,A -85,B 0,C 180,E1 -12898.008,E2 -12898.008} C_VEL
LIN {X 0,Y 372.912,Z 309.644,A -85,B 0,C 180,E1 -12898.678,E2 -12898.678} C_VEL
LIN {X 0,Y 371.423,Z 301.132,A -85,B 0,C 180,E1 -12899.363,E2 -12899.363} C_VEL
LIN {X 0,Y 369.138,Z 291.675,A -85,B 0,C 180,E1 -12899.995,E2 -12899.995} C_VEL
LIN {X 0,Y 367.902,Z 286.982,A -85,B 0,C 180,E1 -12900.292,E2 -12900.292} C_VEL
LIN {X 0,Y 367.919,Z 285.476,A -85,B 0,C 180,E1 -12901.652,E2 -12901.652} C_VEL
LIN {X 0,Y 367.281,Z 284.564,A -85,B 0,C 180,E1 -12902.555,E2 -12902.555} C_VEL
LIN {X 0,Y 364.449,Z 283.314,A -85,B 0,C 180,E1 -12904.031,E2 -12904.031} C_VEL
LIN {X 0,Y 362.07,Z 282.342,A -85,B 0,C 180,E1 -12905.225,E2 -12905.225} C_VEL
LIN {X 0,Y 361.097,Z 281.508,A -85,B 0,C 180,E1 -12906.146,E2 -12906.146} C_VEL
LIN {X 0,Y 361.044,Z 281.193,A -85,B 0,C 180,E1 -12906.457,E2 -12906.457} C_VEL
LIN {X 0,Y 361.285,Z 277.597,A -85,B 0,C 180,E1 -12909.934,E2 -12909.934} C_VEL
LIN {X 0,Y 361.47,Z 274.645,A -85,B 0,C 180,E1 -12912.88,E2 -12912.88} C_VEL
LIN {X 0,Y 361.584,Z 272.255,A -85,B 0,C 180,E1 -12915.599,E2 -12915.599} C_VEL
LIN {X 0,Y 361.772,Z 272.235,A -85,B 0,C 180,E1 -12918.665,E2 -12918.665} C_VEL
LIN {X 0,Y 361.853,Z 272.227,A -85,B 0,C 180,E1 -12921.577,E2 -12921.577} C_VEL
LIN {X 0,Y 361.855,Z 272.226,A -85,B 0,C 180,E1 -12924.656,E2 -12924.656} C_VEL
LIN {X 0,Y 361.819,Z 272.228,A -85,B 0,C 180,E1 -12928.372,E2 -12928.372} C_VEL
LIN {X 0,Y 361.89,Z 272.222,A -85,B 0,C 180,E1 -12932.222,E2 -12932.222} C_VEL
LIN {X 0,Y 361.909,Z 272.217,A -85,B 0,C 180,E1 -12934.711,E2 -12934.711} C_VEL
LIN {X 0,Y 361.864,Z 272.224,A -85,B 0,C 180,E1 -12938.348,E2 -12938.348} C_VEL
LIN {X 0,Y 361.952,Z 272.208,A -85,B 0,C 180,E1 -12942.063,E2 -12942.063} C_VEL
LIN {X 0,Y 361.984,Z 272.204,A -85,B 0,C 180,E1 -12946.103,E2 -12946.103} C_VEL
LIN {X 0,Y 362.022,Z 272.2,A -85,B 0,C 180,E1 -12949.94,E2 -12949.94} C_VEL
LIN {X 0,Y 362.122,Z 272.185,A -85,B 0,C 180,E1 -12953.315,E2 -12953.315} C_VEL
LIN {X 0,Y 362.272,Z 272.168,A -85,B 0,C 180,E1 -12957.778,E2 -12957.778} C_VEL
LIN {X 0,Y 362.416,Z 272.153,A -85,B 0,C 180,E1 -12960.002,E2 -12960.002} C_VEL
LIN {X 0,Y 362.269,Z 272.169,A -85,B 0,C 180,E1 -12962.226,E2 -12962.226} C_VEL
LIN {X 0,Y 362.162,Z 272.181,A -85,B 0,C 180,E1 -12966.688,E2 -12966.688} C_VEL
LIN {X 0,Y 362.065,Z 272.198,A -85,B 0,C 180,E1 -12968.935,E2 -12968.935} C_VEL
LIN {X 0,Y 361.956,Z 272.211,A -85,B 0,C 180,E1 -12972.334,E2 -12972.334} C_VEL
LIN {X 0,Y 361.954,Z 272.212,A -85,B 0,C 180,E1 -12974.622,E2 -12974.622} C_VEL
LIN {X 0,Y 361.949,Z 272.214,A -85,B 0,C 180,E1 -12978.102,E2 -12978.102} C_VEL
LIN {X 0,Y 361.853,Z 272.224,A -85,B 0,C 180,E1 -12981.657,E2 -12981.657} C_VEL
LIN {X 0,Y 361.887,Z 272.22,A -85,B 0,C 180,E1 -12985.295,E2 -12985.295} C_VEL
LIN {X 0,Y 361.849,Z 272.23,A -85,B 0,C 180,E1 -12989.076,E2 -12989.076} C_VEL
LIN {X 0,Y 361.843,Z 272.23,A -85,B 0,C 180,E1 -12992.947,E2 -12992.947} C_VEL
LIN {X 0,Y 361.863,Z 272.228,A -85,B 0,C 180,E1 -12995.639,E2 -12995.639} C_VEL
LIN {X 0,Y 361.869,Z 272.225,A -85,B 0,C 180,E1 -12999.029,E2 -12999.029} C_VEL
LIN {X 0,Y 361.853,Z 272.226,A -85,B 0,C 180,E1 -13002.438,E2 -13002.438} C_VEL
LIN {X 0,Y 361.814,Z 272.228,A -85,B 0,C 180,E1 -13005.949,E2 -13005.949} C_VEL
LIN {X 0,Y 361.843,Z 272.288,A -85,B 0,C 180,E1 -13008.116,E2 -13008.116} C_VEL
LIN {X 0,Y 362.58,Z 276.151,A -85,B 0,C 180,E1 -13010.837,E2 -13010.837} C_VEL
LIN {X 0,Y 363.511,Z 281.842,A -85,B 0,C 180,E1 -13014.551,E2 -13014.551} C_VEL
LIN {X 0,Y 363.837,Z 284.438,A -85,B 0,C 180,E1 -13016.163,E2 -13016.163} C_VEL
LIN {X 0,Y 363.596,Z 288.077,A -85,B 0,C 180,E1 -13018.266,E2 -13018.266} C_VEL
LIN {X 0,Y 362.78,Z 294.242,A -85,B 0,C 180,E1 -13021.667,E2 -13021.667} C_VEL
LIN {X 0,Y 362.041,Z 301.154,A -85,B 0,C 180,E1 -13025.334,E2 -13025.334} C_VEL
LIN {X 0,Y 361.304,Z 309.264,A -85,B 0,C 180,E1 -13029.506,E2 -13029.506} C_VEL
LIN {X 0,Y 360.927,Z 316.271,A -85,B 0,C 180,E1 -13033.019,E2 -13033.019} C_VEL
LIN {X 0,Y 360.919,Z 317.155,A -85,B 0,C 180,E1 -13033.347,E2 -13033.347} C_VEL
LIN {X 0,Y 363.025,Z 329.155,A -85,B 0,C 180,E1 -13033.988,E2 -13033.988} C_VEL
LIN {X 0,Y 364.262,Z 339.536,A -85,B 0,C 180,E1 -13034.732,E2 -13034.732} C_VEL
LIN {X 0,Y 364.684,Z 348.262,A -85,B 0,C 180,E1 -13035.493,E2 -13035.493} C_VEL
LIN {X 0,Y 364.314,Z 355.169,A -85,B 0,C 180,E1 -13036.19,E2 -13036.19} C_VEL
LIN {X 0,Y 363.411,Z 363.136,A -85,B 0,C 180,E1 -13037.152,E2 -13037.152} C_VEL
LIN {X 0,Y 362.777,Z 368.882,A -85,B 0,C 180,E1 -13037.981,E2 -13037.981} C_VEL
LIN {X 0,Y 362.109,Z 375.308,A -85,B 0,C 180,E1 -13039.094,E2 -13039.094} C_VEL
LIN {X 0,Y 361.553,Z 380.665,A -85,B 0,C 180,E1 -13040.209,E2 -13040.209} C_VEL
LIN {X 0,Y 360.995,Z 386.112,A -85,B 0,C 180,E1 -13041.606,E2 -13041.606} C_VEL
LIN {X 0,Y 360.705,Z 389.67,A -85,B 0,C 180,E1 -13042.726,E2 -13042.726} C_VEL
LIN {X 0,Y 360.438,Z 393.769,A -85,B 0,C 180,E1 -13044.407,E2 -13044.407} C_VEL
LIN {X 0,Y 360.425,Z 395.8,A -85,B 0,C 180,E1 -13045.528,E2 -13045.528} C_VEL
LIN {X 0,Y 360.346,Z 397.325,A -85,B 0,C 180,E1 -13046.647,E2 -13046.647} C_VEL
LIN {X 0,Y 360.356,Z 398.311,A -85,B 0,C 180,E1 -13047.766,E2 -13047.766} C_VEL
LIN {X 0,Y 360.455,Z 398.725,A -85,B 0,C 180,E1 -13048.884,E2 -13048.884} C_VEL
LIN {X 0,Y 360.479,Z 398.67,A -85,B 0,C 180,E1 -13050.001,E2 -13050.001} C_VEL
LIN {X 0,Y 360.477,Z 398.151,A -85,B 0,C 180,E1 -13051.119,E2 -13051.119} C_VEL
LIN {X 0,Y 360.403,Z 397.141,A -85,B 0,C 180,E1 -13052.237,E2 -13052.237} C_VEL
LIN {X 0,Y 360.411,Z 394.507,A -85,B 0,C 180,E1 -13053.915,E2 -13053.915} C_VEL
LIN {X 0,Y 360.461,Z 392.121,A -85,B 0,C 180,E1 -13055.035,E2 -13055.035} C_VEL
LIN {X 0,Y 360.594,Z 387.208,A -85,B 0,C 180,E1 -13056.717,E2 -13056.717} C_VEL
LIN {X 0,Y 360.799,Z 383.103,A -85,B 0,C 180,E1 -13057.838,E2 -13057.838} C_VEL
LIN {X 0,Y 361.067,Z 378.152,A -85,B 0,C 180,E1 -13058.96,E2 -13058.96} C_VEL
LIN {X 0,Y 361.412,Z 372.176,A -85,B 0,C 180,E1 -13060.081,E2 -13060.081} C_VEL
LIN {X 0,Y 361.909,Z 364.901,A -85,B 0,C 180,E1 -13061.199,E2 -13061.199} C_VEL
LIN {X 0,Y 362.43,Z 357.126,A -85,B 0,C 180,E1 -13062.175,E2 -13062.175} C_VEL
LIN {X 0,Y 362.959,Z 350.471,A -85,B 0,C 180,E1 -13062.868,E2 -13062.868} C_VEL
LIN {X 0,Y 362.784,Z 342.513,A -85,B 0,C 180,E1 -13063.565,E2 -13063.565} C_VEL
LIN {X 0,Y 362.081,Z 333.126,A -85,B 0,C 180,E1 -13064.224,E2 -13064.224} C_VEL
LIN {X 0,Y 361.192,Z 323.318,A -85,B 0,C 180,E1 -13064.744,E2 -13064.744} C_VEL
LIN {X 0,Y 360.632,Z 317.369,A -85,B 0,C 180,E1 -13065.002,E2 -13065.002} C_VEL
LIN {X 0,Y 360.919,Z 309.635,A -85,B 0,C 180,E1 -13068.743,E2 -13068.743} C_VEL
LIN {X 0,Y 361.362,Z 302.374,A -85,B 0,C 180,E1 -13072.288,E2 -13072.288} C_VEL
LIN {X 0,Y 361.9,Z 295.103,A -85,B 0,C 180,E1 -13075.91,E2 -13075.91} C_VEL
LIN {X 0,Y 362.5,Z 288.538,A -85,B 0,C 180,E1 -13079.254,E2 -13079.254} C_VEL
LIN {X 0,Y 363.108,Z 282.953,A -85,B 0,C 180,E1 -13082.159,E2 -13082.159} C_VEL
LIN {X 0,Y 363.124,Z 279.28,A -85,B 0,C 180,E1 -13084.145,E2 -13084.145} C_VEL
LIN {X 0,Y 362.189,Z 273.784,A -85,B 0,C 180,E1 -13087.289,E2 -13087.289} C_VEL
LIN {X 0,Y 361.947,Z 272.214,A -85,B 0,C 180,E1 -13088.265,E2 -13088.265} C_VEL
LIN {X 0,Y 361.846,Z 272.224,A -85,B 0,C 180,E1 -13092.432,E2 -13092.432} C_VEL
LIN {X 0,Y 361.828,Z 272.229,A -85,B 0,C 180,E1 -13095.947,E2 -13095.947} C_VEL
LIN {X 0,Y 361.844,Z 272.223,A -85,B 0,C 180,E1 -13099.245,E2 -13099.245} C_VEL
LIN {X 0,Y 361.872,Z 272.219,A -85,B 0,C 180,E1 -13102.777,E2 -13102.777} C_VEL
LIN {X 0,Y 361.864,Z 272.225,A -85,B 0,C 180,E1 -13105.719,E2 -13105.719} C_VEL
LIN {X 0,Y 361.885,Z 272.222,A -85,B 0,C 180,E1 -13109.671,E2 -13109.671} C_VEL
LIN {X 0,Y 361.964,Z 272.212,A -85,B 0,C 180,E1 -13113.474,E2 -13113.474} C_VEL
LIN {X 0,Y 361.892,Z 272.221,A -85,B 0,C 180,E1 -13117.143,E2 -13117.143} C_VEL
LIN {X 0,Y 361.895,Z 272.218,A -85,B 0,C 180,E1 -13120.721,E2 -13120.721} C_VEL
LIN {X 0,Y 361.952,Z 272.209,A -85,B 0,C 180,E1 -13124.225,E2 -13124.225} C_VEL
LIN {X 0,Y 362.008,Z 272.204,A -85,B 0,C 180,E1 -13126.526,E2 -13126.526} C_VEL
LIN {X 0,Y 362.008,Z 272.202,A -85,B 0,C 180,E1 -13129.936,E2 -13129.936} C_VEL
LIN {X 0,Y 362.156,Z 272.185,A -85,B 0,C 180,E1 -13133.312,E2 -13133.312} C_VEL
LIN {X 0,Y 362.287,Z 272.167,A -85,B 0,C 180,E1 -13137.775,E2 -13137.775} C_VEL
LIN {X 0,Y 362.432,Z 272.15,A -85,B 0,C 180,E1 -13139.998,E2 -13139.998} C_VEL
LIN {X 0,Y 362.289,Z 272.17,A -85,B 0,C 180,E1 -13142.221,E2 -13142.221} C_VEL
LIN {X 0,Y 362.177,Z 272.184,A -85,B 0,C 180,E1 -13146.684,E2 -13146.684} C_VEL
LIN {X 0,Y 362.078,Z 272.194,A -85,B 0,C 180,E1 -13148.931,E2 -13148.931} C_VEL
LIN {X 0,Y 361.964,Z 272.212,A -85,B 0,C 180,E1 -13152.33,E2 -13152.33} C_VEL
LIN {X 0,Y 361.965,Z 272.21,A -85,B 0,C 180,E1 -13154.618,E2 -13154.618} C_VEL
LIN {X 0,Y 361.959,Z 272.213,A -85,B 0,C 180,E1 -13158.097,E2 -13158.097} C_VEL
LIN {X 0,Y 361.892,Z 272.22,A -85,B 0,C 180,E1 -13161.65,E2 -13161.65} C_VEL
LIN {X 0,Y 361.928,Z 272.213,A -85,B 0,C 180,E1 -13165.287,E2 -13165.287} C_VEL
LIN {X 0,Y 361.907,Z 272.219,A -85,B 0,C 180,E1 -13167.776,E2 -13167.776} C_VEL
LIN {X 0,Y 361.835,Z 272.229,A -85,B 0,C 180,E1 -13171.627,E2 -13171.627} C_VEL
LIN {X 0,Y 361.87,Z 272.223,A -85,B 0,C 180,E1 -13175.342,E2 -13175.342} C_VEL
LIN {X 0,Y 361.869,Z 272.222,A -85,B 0,C 180,E1 -13179.025,E2 -13179.025} C_VEL
LIN {X 0,Y 361.88,Z 272.218,A -85,B 0,C 180,E1 -13182.438,E2 -13182.438} C_VEL
LIN {X 0,Y 361.921,Z 272.214,A -85,B 0,C 180,E1 -13185.926,E2 -13185.926} C_VEL
LIN {X 0,Y 361.896,Z 272.221,A -85,B 0,C 180,E1 -13189.229,E2 -13189.229} C_VEL
LIN {X 0,Y 361.859,Z 272.225,A -85,B 0,C 180,E1 -13192.98,E2 -13192.98} C_VEL
LIN {X 0,Y 361.847,Z 272.225,A -85,B 0,C 180,E1 -13196.628,E2 -13196.628} C_VEL
LIN {X 0,Y 361.864,Z 272.22,A -85,B 0,C 180,E1 -13199.67,E2 -13199.67} C_VEL
LIN {X 0,Y 361.941,Z 272.211,A -85,B 0,C 180,E1 -13203.473,E2 -13203.473} C_VEL
LIN {X 0,Y 361.888,Z 272.218,A -85,B 0,C 180,E1 -13207.143,E2 -13207.143} C_VEL
LIN {X 0,Y 361.88,Z 272.218,A -85,B 0,C 180,E1 -13209.537,E2 -13209.537} C_VEL
LIN {X 0,Y 361.639,Z 272.249,A -85,B 0,C 180,E1 -13213.05,E2 -13213.05} C_VEL
LIN {X 0,Y 361.273,Z 272.581,A -85,B 0,C 180,E1 -13216.499,E2 -13216.499} C_VEL
LIN {X 0,Y 361.076,Z 276.312,A -85,B 0,C 180,E1 -13219.91,E2 -13219.91} C_VEL
LIN {X 0,Y 361.159,Z 280.067,A -85,B 0,C 180,E1 -13223.294,E2 -13223.294} C_VEL
LIN {X 0,Y 360.983,Z 283.912,A -85,B 0,C 180,E1 -13226.65,E2 -13226.65} C_VEL
LIN {X 0,Y 360.814,Z 286.887,A -85,B 0,C 180,E1 -13229.162,E2 -13229.162} C_VEL
LIN {X 0,Y 362.55,Z 297.796,A -85,B 0,C 180,E1 -13229.721,E2 -13229.721} C_VEL
LIN {X 0,Y 363.809,Z 305.95,A -85,B 0,C 180,E1 -13230.275,E2 -13230.275} C_VEL
LIN {X 0,Y 363.623,Z 314.575,A -85,B 0,C 180,E1 -13230.968,E2 -13230.968} C_VEL
LIN {X 0,Y 363.1,Z 322.928,A -85,B 0,C 180,E1 -13231.801,E2 -13231.801} C_VEL
LIN {X 0,Y 362.582,Z 330.824,A -85,B 0,C 180,E1 -13232.776,E2 -13232.776} C_VEL
LIN {X 0,Y 362.075,Z 338.196,A -85,B 0,C 180,E1 -13233.894,E2 -13233.894} C_VEL
LIN {X 0,Y 361.53,Z 345.676,A -85,B 0,C 180,E1 -13235.297,E2 -13235.297} C_VEL
LIN {X 0,Y 361.253,Z 351.515,A -85,B 0,C 180,E1 -13236.702,E2 -13236.702} C_VEL
LIN {X 0,Y 360.969,Z 355.35,A -85,B 0,C 180,E1 -13237.832,E2 -13237.832} C_VEL
LIN {X 0,Y 360.619,Z 359.735,A -85,B 0,C 180,E1 -13239.534,E2 -13239.534} C_VEL
LIN {X 0,Y 360.437,Z 362.802,A -85,B 0,C 180,E1 -13241.242,E2 -13241.242} C_VEL
LIN {X 0,Y 360.361,Z 364.554,A -85,B 0,C 180,E1 -13242.819,E2 -13242.819} C_VEL
LIN {X 0,Y 360.318,Z 365.394,A -85,B 0,C 180,E1 -13244.687,E2 -13244.687} C_VEL
